LIN {X 0,Y 228.554,Z 405.474,A -85,B 0,C 180,E1 -19981.761,E2 -19981.761} C_VEL
LIN {X 0,Y 228.355,Z 405.527,A -85,B 0,C 180,E1 -19987.07,E2 -19987.07} C_VEL
LIN {X 0,Y 228.163,Z 405.519,A -85,B 0,C 180,E1 -19990.649,E2 -19990.649} C_VEL
LIN {X 0,Y 228.064,Z 405.576,A -85,B 0,C 180,E1 -19994.271,E2 -19994.271} C_VEL
LIN {X 0,Y 228.002,Z 405.55,A -85,B 0,C 180,E1 -19997.952,E2 -19997.952} C_VEL
LIN {X 0,Y 227.929,Z 405.587,A -85,B 0,C 180,E1 -20002.328,E2 -20002.328} C_VEL
LIN {X 0,Y 227.94,Z 405.561,A -85,B 0,C 180,E1 -20006.601,E2 -20006.601} C_VEL
LIN {X 0,Y 227.895,Z 405.594,A -85,B 0,C 180,E1 -20010.29,E2 -20010.29} C_VEL
LIN {X 0,Y 227.887,Z 405.574,A -85,B 0,C 180,E1 -20013.717,E2 -20013.717} C_VEL
LIN {X 0,Y 227.868,Z 405.602,A -85,B 0,C 180,E1 -20018.085,E2 -20018.085} C_VEL
LIN {X 0,Y 227.813,Z 405.604,A -85,B 0,C 180,E1 -20022.74,E2 -20022.74} C_VEL
LIN {X 0,Y 227.812,Z 405.544,A -85,B 0,C 180,E1 -20027.258,E2 -20027.258} C_VEL
LIN {X 0,Y 227.868,Z 405.602,A -85,B 0,C 180,E1 -20031.913,E2 -20031.913} C_VEL
LIN {X 0,Y 227.951,Z 405.9,A -85,B 0,C 180,E1 -20032.927,E2 -20032.927} C_VEL
LIN {X 0,Y 228.325,Z 407.207,A -85,B 0,C 180,E1 -20033.243,E2 -20033.243} C_VEL
LIN {X 0,Y 229.944,Z 409.725,A -85,B 0,C 180,E1 -20033.653,E2 -20033.653} C_VEL
LIN {X 0,Y 238.782,Z 424.968,A -85,B 0,C 180,E1 -20035.756,E2 -20035.756} C_VEL
LIN {X 0,Y 245.467,Z 437.776,A -85,B 0,C 180,E1 -20037.257,E2 -20037.257} C_VEL
LIN {X 0,Y 252.292,Z 450.513,A -85,B 0,C 180,E1 -20038.673,E2 -20038.673} C_VEL
LIN {X 0,Y 260.836,Z 463.188,A -85,B 0,C 180,E1 -20040.213,E2 -20040.213} C_VEL
LIN {X 0,Y 271.083,Z 475.491,A -85,B 0,C 180,E1 -20041.818,E2 -20041.818} C_VEL
LIN {X 0,Y 285.472,Z 490.143,A -85,B 0,C 180,E1 -20043.771,E2 -20043.771} C_VEL
LIN {X 0,Y 299.445,Z 502.11,A -85,B 0,C 180,E1 -20045.429,E2 -20045.429} C_VEL
LIN {X 0,Y 307.354,Z 508.55,A -85,B 0,C 180,E1 -20046.449,E2 -20046.449} C_VEL
LIN {X 0,Y 315.809,Z 515.11,A -85,B 0,C 180,E1 -20047.77,E2 -20047.77} C_VEL
LIN {X 0,Y 323.821,Z 521.078,A -85,B 0,C 180,E1 -20049.216,E2 -20049.216} C_VEL
LIN {X 0,Y 332.128,Z 527.32,A -85,B 0,C 180,E1 -20050.94,E2 -20050.94} C_VEL
LIN {X 0,Y 338.952,Z 531.879,A -85,B 0,C 180,E1 -20052.51,E2 -20052.51} C_VEL
LIN {X 0,Y 345.131,Z 536.469,A -85,B 0,C 180,E1 -20054.129,E2 -20054.129} C_VEL
LIN {X 0,Y 348.902,Z 539.004,A -85,B 0,C 180,E1 -20055.208,E2 -20055.208} C_VEL
LIN {X 0,Y 353.812,Z 541.898,A -85,B 0,C 180,E1 -20056.731,E2 -20056.731} C_VEL
LIN {X 0,Y 357.273,Z 544.165,A -85,B 0,C 180,E1 -20057.966,E2 -20057.966} C_VEL
LIN {X 0,Y 361.925,Z 547.614,A -85,B 0,C 180,E1 -20059.935,E2 -20059.935} C_VEL
LIN {X 0,Y 364.433,Z 549.121,A -85,B 0,C 180,E1 -20061.125,E2 -20061.125} C_VEL
LIN {X 0,Y 368.054,Z 551.052,A -85,B 0,C 180,E1 -20063.181,E2 -20063.181} C_VEL
LIN {X 0,Y 369.976,Z 551.886,A -85,B 0,C 180,E1 -20064.55,E2 -20064.55} C_VEL
LIN {X 0,Y 371.247,Z 552.35,A -85,B 0,C 180,E1 -20065.657,E2 -20065.657} C_VEL
LIN {X 0,Y 372.237,Z 552.641,A -85,B 0,C 180,E1 -20066.753,E2 -20066.753} C_VEL
LIN {X 0,Y 372.88,Z 552.99,A -85,B 0,C 180,E1 -20067.839,E2 -20067.839} C_VEL
LIN {X 0,Y 373.24,Z 553.258,A -85,B 0,C 180,E1 -20068.921,E2 -20068.921} C_VEL
LIN {X 0,Y 373.406,Z 553.214,A -85,B 0,C 180,E1 -20070,E2 -20070} C_VEL
LIN {X 0,Y 373.262,Z 553.193,A -85,B 0,C 180,E1 -20071.079,E2 -20071.079} C_VEL
LIN {X 0,Y 372.799,Z 552.913,A -85,B 0,C 180,E1 -20072.373,E2 -20072.373} C_VEL
LIN {X 0,Y 371.244,Z 552.366,A -85,B 0,C 180,E1 -20074.342,E2 -20074.342} C_VEL
LIN {X 0,Y 369.973,Z 551.918,A -85,B 0,C 180,E1 -20075.45,E2 -20075.45} C_VEL
LIN {X 0,Y 368.059,Z 551.052,A -85,B 0,C 180,E1 -20076.825,E2 -20076.825} C_VEL
LIN {X 0,Y 364.441,Z 549.115,A -85,B 0,C 180,E1 -20078.874,E2 -20078.874} C_VEL
LIN {X 0,Y 360.218,Z 546.455,A -85,B 0,C 180,E1 -20080.812,E2 -20080.812} C_VEL
LIN {X 0,Y 355.924,Z 543.055,A -85,B 0,C 180,E1 -20082.544,E2 -20082.544} C_VEL
LIN {X 0,Y 351.923,Z 540.864,A -85,B 0,C 180,E1 -20083.865,E2 -20083.865} C_VEL
LIN {X 0,Y 345.74,Z 536.848,A -85,B 0,C 180,E1 -20085.708,E2 -20085.708} C_VEL
LIN {X 0,Y 338.968,Z 531.895,A -85,B 0,C 180,E1 -20087.498,E2 -20087.498} C_VEL
LIN {X 0,Y 331.843,Z 527.13,A -85,B 0,C 180,E1 -20089.121,E2 -20089.121} C_VEL
LIN {X 0,Y 323.739,Z 521.021,A -85,B 0,C 180,E1 -20090.798,E2 -20090.798} C_VEL
LIN {X 0,Y 315.796,Z 515.105,A -85,B 0,C 180,E1 -20092.23,E2 -20092.23} C_VEL
LIN {X 0,Y 307.554,Z 508.722,A -85,B 0,C 180,E1 -20093.524,E2 -20093.524} C_VEL
LIN {X 0,Y 300.572,Z 502.979,A -85,B 0,C 180,E1 -20094.436,E2 -20094.436} C_VEL
LIN {X 0,Y 291.164,Z 495.16,A -85,B 0,C 180,E1 -20095.539,E2 -20095.539} C_VEL
LIN {X 0,Y 280.858,Z 485.585,A -85,B 0,C 180,E1 -20096.826,E2 -20096.826} C_VEL
LIN {X 0,Y 268.674,Z 472.809,A -85,B 0,C 180,E1 -20098.54,E2 -20098.54} C_VEL
LIN {X 0,Y 260.028,Z 462.067,A -85,B 0,C 180,E1 -20099.925,E2 -20099.925} C_VEL
LIN {X 0,Y 252.005,Z 450.092,A -85,B 0,C 180,E1 -20101.38,E2 -20101.38} C_VEL
LIN {X 0,Y 245.113,Z 437.01,A -85,B 0,C 180,E1 -20102.822,E2 -20102.822} C_VEL
LIN {X 0,Y 237.86,Z 423.227,A -85,B 0,C 180,E1 -20104.459,E2 -20104.459} C_VEL
LIN {X 0,Y 229.958,Z 409.757,A -85,B 0,C 180,E1 -20106.343,E2 -20106.343} C_VEL
LIN {X 0,Y 228.326,Z 407.225,A -85,B 0,C 180,E1 -20106.756,E2 -20106.756} C_VEL
LIN {X 0,Y 227.923,Z 405.904,A -85,B 0,C 180,E1 -20107.08,E2 -20107.08} C_VEL
LIN {X 0,Y 227.865,Z 405.602,A -85,B 0,C 180,E1 -20108.086,E2 -20108.086} C_VEL
LIN {X 0,Y 227.81,Z 405.544,A -85,B 0,C 180,E1 -20112.741,E2 -20112.741} C_VEL
LIN {X 0,Y 227.893,Z 405.594,A -85,B 0,C 180,E1 -20117.278,E2 -20117.278} C_VEL
LIN {X 0,Y 227.866,Z 405.603,A -85,B 0,C 180,E1 -20121.915,E2 -20121.915} C_VEL
LIN {X 0,Y 227.885,Z 405.575,A -85,B 0,C 180,E1 -20126.373,E2 -20126.373} C_VEL
LIN {X 0,Y 227.914,Z 405.582,A -85,B 0,C 180,E1 -20130.438,E2 -20130.438} C_VEL
LIN {X 0,Y 227.923,Z 405.575,A -85,B 0,C 180,E1 -20134.426,E2 -20134.426} C_VEL
LIN {X 0,Y 227.957,Z 405.575,A -85,B 0,C 180,E1 -20138.288,E2 -20138.288} C_VEL
LIN {X 0,Y 228.03,Z 405.558,A -85,B 0,C 180,E1 -20142.827,E2 -20142.827} C_VEL
LIN {X 0,Y 228.09,Z 405.55,A -85,B 0,C 180,E1 -20147.545,E2 -20147.545} C_VEL
LIN {X 0,Y 228.301,Z 405.507,A -85,B 0,C 180,E1 -20151.147,E2 -20151.147} C_VEL
LIN {X 0,Y 228.351,Z 405.527,A -85,B 0,C 180,E1 -20152.929,E2 -20152.929} C_VEL
LIN {X 0,Y 228.551,Z 405.475,A -85,B 0,C 180,E1 -20158.239,E2 -20158.239} C_VEL
LIN {X 0,Y 228.551,Z 405.487,A -85,B 0,C 180,E1 -20161.763,E2 -20161.763} C_VEL
LIN {X 0,Y 228.352,Z 405.514,A -85,B 0,C 180,E1 -20167.073,E2 -20167.073} C_VEL
LIN {X 0,Y 228.16,Z 405.522,A -85,B 0,C 180,E1 -20170.651,E2 -20170.651} C_VEL
LIN {X 0,Y 228.062,Z 405.574,A -85,B 0,C 180,E1 -20174.273,E2 -20174.273} C_VEL
LIN {X 0,Y 228,Z 405.541,A -85,B 0,C 180,E1 -20177.954,E2 -20177.954} C_VEL
LIN {X 0,Y 227.928,Z 405.59,A -85,B 0,C 180,E1 -20182.331,E2 -20182.331} C_VEL
LIN {X 0,Y 227.941,Z 405.556,A -85,B 0,C 180,E1 -20186.604,E2 -20186.604} C_VEL
LIN {X 0,Y 227.908,Z 405.597,A -85,B 0,C 180,E1 -20190.298,E2 -20190.298} C_VEL
LIN {X 0,Y 227.888,Z 405.571,A -85,B 0,C 180,E1 -20193.72,E2 -20193.72} C_VEL
LIN {X 0,Y 227.871,Z 405.595,A -85,B 0,C 180,E1 -20198.087,E2 -20198.087} C_VEL
LIN {X 0,Y 227.917,Z 405.593,A -85,B 0,C 180,E1 -20202.719,E2 -20202.719} C_VEL
LIN {X 0,Y 227.899,Z 405.809,A -85,B 0,C 180,E1 -20207.645,E2 -20207.645} C_VEL
LIN {X 0,Y 229.638,Z 413.101,A -85,B 0,C 180,E1 -20212.26,E2 -20212.26} C_VEL
LIN {X 0,Y 230.148,Z 415.394,A -85,B 0,C 180,E1 -20213.453,E2 -20213.453} C_VEL
LIN {X 0,Y 232.024,Z 419.408,A -85,B 0,C 180,E1 -20214.009,E2 -20214.009} C_VEL
LIN {X 0,Y 240.511,Z 437.365,A -85,B 0,C 180,E1 -20216.088,E2 -20216.088} C_VEL
LIN {X 0,Y 243.824,Z 445.896,A -85,B 0,C 180,E1 -20216.9,E2 -20216.9} C_VEL
LIN {X 0,Y 247.873,Z 469.061,A -85,B 0,C 180,E1 -20218.278,E2 -20218.278} C_VEL
LIN {X 0,Y 248.138,Z 472.35,A -85,B 0,C 180,E1 -20218.425,E2 -20218.425} C_VEL
LIN {X 0,Y 248.05,Z 474.394,A -85,B 0,C 180,E1 -20218.48,E2 -20218.48} C_VEL
LIN {X 0,Y 247.227,Z 480.242,A -85,B 0,C 180,E1 -20218.559,E2 -20218.559} C_VEL
LIN {X 0,Y 241.567,Z 499.251,A -85,B 0,C 180,E1 -20218.392,E2 -20218.392} C_VEL
LIN {X 0,Y 240.81,Z 505.095,A -85,B 0,C 180,E1 -20218.482,E2 -20218.482} C_VEL
LIN {X 0,Y 239.876,Z 524.739,A -85,B 0,C 180,E1 -20219.12,E2 -20219.12} C_VEL
LIN {X 0,Y 238.394,Z 538.868,A -85,B 0,C 180,E1 -20219.924,E2 -20219.924} C_VEL
LIN {X 0,Y 236.942,Z 548.514,A -85,B 0,C 180,E1 -20220.699,E2 -20220.699} C_VEL
LIN {X 0,Y 235.223,Z 558.034,A -85,B 0,C 180,E1 -20221.686,E2 -20221.686} C_VEL
LIN {X 0,Y 233.004,Z 568.622,A -85,B 0,C 180,E1 -20223.101,E2 -20223.101} C_VEL
LIN {X 0,Y 230.914,Z 577.345,A -85,B 0,C 180,E1 -20224.54,E2 -20224.54} C_VEL
LIN {X 0,Y 229.001,Z 584.763,A -85,B 0,C 180,E1 -20226.007,E2 -20226.007} C_VEL
LIN {X 0,Y 226.579,Z 593.556,A -85,B 0,C 180,E1 -20228.149,E2 -20228.149} C_VEL
LIN {X 0,Y 225.092,Z 599.552,A -85,B 0,C 180,E1 -20229.914,E2 -20229.914} C_VEL
LIN {X 0,Y 223.198,Z 605.86,A -85,B 0,C 180,E1 -20232.122,E2 -20232.122} C_VEL
LIN {X 0,Y 221.656,Z 611.133,A -85,B 0,C 180,E1 -20234.366,E2 -20234.366} C_VEL
LIN {X 0,Y 220.226,Z 616.228,A -85,B 0,C 180,E1 -20237.093,E2 -20237.093} C_VEL
LIN {X 0,Y 219.318,Z 620.197,A -85,B 0,C 180,E1 -20239.849,E2 -20239.849} C_VEL
LIN {X 0,Y 218.762,Z 623.136,A -85,B 0,C 180,E1 -20242.617,E2 -20242.617} C_VEL
LIN {X 0,Y 218.572,Z 624.64,A -85,B 0,C 180,E1 -20244.465,E2 -20244.465} C_VEL
LIN {X 0,Y 218.525,Z 626.171,A -85,B 0,C 180,E1 -20248.158,E2 -20248.158} C_VEL
LIN {X 0,Y 218.622,Z 626.454,A -85,B 0,C 180,E1 -20250.001,E2 -20250.001} C_VEL
LIN {X 0,Y 218.501,Z 625.572,A -85,B 0,C 180,E1 -20253.689,E2 -20253.689} C_VEL
LIN {X 0,Y 218.568,Z 624.64,A -85,B 0,C 180,E1 -20255.536,E2 -20255.536} C_VEL
LIN {X 0,Y 219.088,Z 621.286,A -85,B 0,C 180,E1 -20259.23,E2 -20259.23} C_VEL
LIN {X 0,Y 219.88,Z 617.656,A -85,B 0,C 180,E1 -20261.991,E2 -20261.991} C_VEL
LIN {X 0,Y 221.07,Z 612.92,A -85,B 0,C 180,E1 -20264.734,E2 -20264.734} C_VEL
LIN {X 0,Y 222.916,Z 606.951,A -85,B 0,C 180,E1 -20267.429,E2 -20267.429} C_VEL
LIN {X 0,Y 224.294,Z 602.171,A -85,B 0,C 180,E1 -20269.209,E2 -20269.209} C_VEL
LIN {X 0,Y 226.087,Z 595.69,A -85,B 0,C 180,E1 -20271.248,E2 -20271.248} C_VEL
LIN {X 0,Y 228.023,Z 588.459,A -85,B 0,C 180,E1 -20273.14,E2 -20273.14} C_VEL
LIN {X 0,Y 230.132,Z 580.635,A -85,B 0,C 180,E1 -20274.829,E2 -20274.829} C_VEL
LIN {X 0,Y 232.114,Z 572.554,A -85,B 0,C 180,E1 -20276.284,E2 -20276.284} C_VEL
LIN {X 0,Y 234.273,Z 562.796,A -85,B 0,C 180,E1 -20277.71,E2 -20277.71} C_VEL
LIN {X 0,Y 235.869,Z 554.406,A -85,B 0,C 180,E1 -20278.716,E2 -20278.716} C_VEL
LIN {X 0,Y 237.601,Z 543.903,A -85,B 0,C 180,E1 -20279.699,E2 -20279.699} C_VEL
LIN {X 0,Y 239.038,Z 533.59,A -85,B 0,C 180,E1 -20280.413,E2 -20280.413} C_VEL
LIN {X 0,Y 239.996,Z 523.576,A -85,B 0,C 180,E1 -20280.917,E2 -20280.917} C_VEL
LIN {X 0,Y 240.908,Z 502.246,A -85,B 0,C 180,E1 -20281.601,E2 -20281.601} C_VEL
LIN {X 0,Y 242.123,Z 471.972,A -85,B 0,C 180,E1 -20282.46,E2 -20282.46} C_VEL
LIN {X 0,Y 238.762,Z 452.033,A -85,B 0,C 180,E1 -20283.673,E2 -20283.673} C_VEL
LIN {X 0,Y 237.532,Z 446.723,A -85,B 0,C 180,E1 -20284.058,E2 -20284.058} C_VEL
LIN {X 0,Y 230.678,Z 430.987,A -85,B 0,C 180,E1 -20285.797,E2 -20285.797} C_VEL
LIN {X 0,Y 224.359,Z 418.419,A -85,B 0,C 180,E1 -20287.454,E2 -20287.454} C_VEL
LIN {X 0,Y 222.822,Z 414.942,A -85,B 0,C 180,E1 -20288.007,E2 -20288.007} C_VEL
LIN {X 0,Y 221.346,Z 408.913,A -85,B 0,C 180,E1 -20291.819,E2 -20291.819} C_VEL
LIN {X 0,Y 220.803,Z 406.564,A -85,B 0,C 180,E1 -20293.486,E2 -20293.486} C_VEL
LIN {X 0,Y 220.863,Z 406.473,A -85,B 0,C 180,E1 -20298.068,E2 -20298.068} C_VEL
LIN {X 0,Y 220.838,Z 406.477,A -85,B 0,C 180,E1 -20302.794,E2 -20302.794} C_VEL
LIN {X 0,Y 220.827,Z 406.456,A -85,B 0,C 180,E1 -20307.244,E2 -20307.244} C_VEL
LIN {X 0,Y 220.839,Z 406.453,A -85,B 0,C 180,E1 -20311.486,E2 -20311.486} C_VEL
LIN {X 0,Y 220.869,Z 406.457,A -85,B 0,C 180,E1 -20315.564,E2 -20315.564} C_VEL
LIN {X 0,Y 220.894,Z 406.441,A -85,B 0,C 180,E1 -20319.513,E2 -20319.513} C_VEL
LIN {X 0,Y 221.018,Z 406.423,A -85,B 0,C 180,E1 -20323.369,E2 -20323.369} C_VEL
LIN {X 0,Y 221.113,Z 406.402,A -85,B 0,C 180,E1 -20329.005,E2 -20329.005} C_VEL
LIN {X 0,Y 221.291,Z 406.388,A -85,B 0,C 180,E1 -20332.701,E2 -20332.701} C_VEL
LIN {X 0,Y 221.513,Z 406.363,A -85,B 0,C 180,E1 -20338.181,E2 -20338.181} C_VEL
LIN {X 0,Y 221.512,Z 406.351,A -85,B 0,C 180,E1 -20341.817,E2 -20341.817} C_VEL
LIN {X 0,Y 221.306,Z 406.402,A -85,B 0,C 180,E1 -20347.297,E2 -20347.297} C_VEL
LIN {X 0,Y 221.112,Z 406.399,A -85,B 0,C 180,E1 -20350.993,E2 -20350.993} C_VEL
LIN {X 0,Y 221.016,Z 406.438,A -85,B 0,C 180,E1 -20356.629,E2 -20356.629} C_VEL
LIN {X 0,Y 220.891,Z 406.435,A -85,B 0,C 180,E1 -20360.485,E2 -20360.485} C_VEL
LIN {X 0,Y 220.866,Z 406.47,A -85,B 0,C 180,E1 -20364.434,E2 -20364.434} C_VEL
LIN {X 0,Y 220.825,Z 406.449,A -85,B 0,C 180,E1 -20368.514,E2 -20368.514} C_VEL
LIN {X 0,Y 220.821,Z 406.465,A -85,B 0,C 180,E1 -20372.754,E2 -20372.754} C_VEL
LIN {X 0,Y 220.836,Z 406.477,A -85,B 0,C 180,E1 -20377.287,E2 -20377.287} C_VEL
LIN {X 0,Y 220.773,Z 406.469,A -85,B 0,C 180,E1 -20381.95,E2 -20381.95} C_VEL
LIN {X 0,Y 220.773,Z 406.442,A -85,B 0,C 180,E1 -20385.546,E2 -20385.546} C_VEL
LIN {X 0,Y 220.807,Z 406.439,A -85,B 0,C 180,E1 -20390.463,E2 -20390.463} C_VEL
LIN {X 0,Y 220.871,Z 406.783,A -85,B 0,C 180,E1 -20391.555,E2 -20391.555} C_VEL
LIN {X 0,Y 221.24,Z 408.118,A -85,B 0,C 180,E1 -20391.887,E2 -20391.887} C_VEL
LIN {X 0,Y 222.989,Z 410.766,A -85,B 0,C 180,E1 -20392.359,E2 -20392.359} C_VEL
LIN {X 0,Y 230.451,Z 423.139,A -85,B 0,C 180,E1 -20394.254,E2 -20394.254} C_VEL
LIN {X 0,Y 237.954,Z 436.997,A -85,B 0,C 180,E1 -20396.05,E2 -20396.05} C_VEL
LIN {X 0,Y 246.373,Z 453.364,A -85,B 0,C 180,E1 -20397.922,E2 -20397.922} C_VEL
LIN {X 0,Y 254.155,Z 465.309,A -85,B 0,C 180,E1 -20399.409,E2 -20399.409} C_VEL
LIN {X 0,Y 261.763,Z 475.126,A -85,B 0,C 180,E1 -20400.699,E2 -20400.699} C_VEL
LIN {X 0,Y 274.478,Z 489.059,A -85,B 0,C 180,E1 -20402.593,E2 -20402.593} C_VEL
LIN {X 0,Y 285.936,Z 499.796,A -85,B 0,C 180,E1 -20404.082,E2 -20404.082} C_VEL
LIN {X 0,Y 296.699,Z 508.846,A -85,B 0,C 180,E1 -20405.365,E2 -20405.365} C_VEL
LIN {X 0,Y 304.926,Z 515.571,A -85,B 0,C 180,E1 -20406.473,E2 -20406.473} C_VEL
LIN {X 0,Y 312.987,Z 521.784,A -85,B 0,C 180,E1 -20407.749,E2 -20407.749} C_VEL
LIN {X 0,Y 321.067,Z 527.71,A -85,B 0,C 180,E1 -20409.205,E2 -20409.205} C_VEL
LIN {X 0,Y 327.826,Z 532.846,A -85,B 0,C 180,E1 -20410.608,E2 -20410.608} C_VEL
LIN {X 0,Y 332.996,Z 536.412,A -85,B 0,C 180,E1 -20411.755,E2 -20411.755} C_VEL
LIN {X 0,Y 338.549,Z 540.283,A -85,B 0,C 180,E1 -20413.104,E2 -20413.104} C_VEL
LIN {X 0,Y 343.97,Z 544.192,A -85,B 0,C 180,E1 -20414.596,E2 -20414.596} C_VEL
LIN {X 0,Y 348.701,Z 547.147,A -85,B 0,C 180,E1 -20416.004,E2 -20416.004} C_VEL
LIN {X 0,Y 352.905,Z 549.493,A -85,B 0,C 180,E1 -20417.371,E2 -20417.371} C_VEL
LIN {X 0,Y 357.622,Z 553.083,A -85,B 0,C 180,E1 -20419.292,E2 -20419.292} C_VEL
LIN {X 0,Y 361.373,Z 555.513,A -85,B 0,C 180,E1 -20421.049,E2 -20421.049} C_VEL
LIN {X 0,Y 363.554,Z 556.729,A -85,B 0,C 180,E1 -20422.223,E2 -20422.223} C_VEL
LIN {X 0,Y 365.443,Z 557.658,A -85,B 0,C 180,E1 -20423.374,E2 -20423.374} C_VEL
LIN {X 0,Y 367.106,Z 558.35,A -85,B 0,C 180,E1 -20424.557,E2 -20424.557} C_VEL
LIN {X 0,Y 368.317,Z 558.822,A -85,B 0,C 180,E1 -20425.622,E2 -20425.622} C_VEL
LIN {X 0,Y 369.338,Z 559.106,A -85,B 0,C 180,E1 -20426.727,E2 -20426.727} C_VEL
LIN {X 0,Y 369.982,Z 559.47,A -85,B 0,C 180,E1 -20427.822,E2 -20427.822} C_VEL
LIN {X 0,Y 370.34,Z 559.737,A -85,B 0,C 180,E1 -20428.912,E2 -20428.912} C_VEL
LIN {X 0,Y 370.526,Z 559.673,A -85,B 0,C 180,E1 -20430,E2 -20430} C_VEL
LIN {X 0,Y 370.373,Z 559.651,A -85,B 0,C 180,E1 -20431.087,E2 -20431.087} C_VEL
LIN {X 0,Y 369.987,Z 559.435,A -85,B 0,C 180,E1 -20432.177,E2 -20432.177} C_VEL
LIN {X 0,Y 369.329,Z 559.095,A -85,B 0,C 180,E1 -20433.272,E2 -20433.272} C_VEL
LIN {X 0,Y 368.306,Z 558.822,A -85,B 0,C 180,E1 -20434.377,E2 -20434.377} C_VEL
LIN {X 0,Y 367.014,Z 558.361,A -85,B 0,C 180,E1 -20435.494,E2 -20435.494} C_VEL
LIN {X 0,Y 365.444,Z 557.664,A -85,B 0,C 180,E1 -20436.626,E2 -20436.626} C_VEL
LIN {X 0,Y 362.347,Z 556.045,A -85,B 0,C 180,E1 -20438.44,E2 -20438.44} C_VEL
LIN {X 0,Y 358.851,Z 553.978,A -85,B 0,C 180,E1 -20440.152,E2 -20440.152} C_VEL
LIN {X 0,Y 354.946,Z 551.149,A -85,B 0,C 180,E1 -20441.817,E2 -20441.817} C_VEL
LIN {X 0,Y 352.841,Z 549.405,A -85,B 0,C 180,E1 -20442.656,E2 -20442.656} C_VEL
LIN {X 0,Y 347.995,Z 546.721,A -85,B 0,C 180,E1 -20444.216,E2 -20444.216} C_VEL
LIN {X 0,Y 343.051,Z 543.53,A -85,B 0,C 180,E1 -20445.664,E2 -20445.664} C_VEL
LIN {X 0,Y 338.092,Z 539.928,A -85,B 0,C 180,E1 -20447.021,E2 -20447.021} C_VEL
LIN {X 0,Y 330.726,Z 534.904,A -85,B 0,C 180,E1 -20448.765,E2 -20448.765} C_VEL
LIN {X 0,Y 323.611,Z 529.586,A -85,B 0,C 180,E1 -20450.289,E2 -20450.289} C_VEL
LIN {X 0,Y 314.843,Z 523.218,A -85,B 0,C 180,E1 -20451.931,E2 -20451.931} C_VEL
LIN {X 0,Y 306.174,Z 516.524,A -85,B 0,C 180,E1 -20453.342,E2 -20453.342} C_VEL
LIN {X 0,Y 298,Z 509.994,A -85,B 0,C 180,E1 -20454.471,E2 -20454.471} C_VEL
LIN {X 0,Y 286.124,Z 499.956,A -85,B 0,C 180,E1 -20455.895,E2 -20455.895} C_VEL
LIN {X 0,Y 276.695,Z 491.195,A -85,B 0,C 180,E1 -20457.106,E2 -20457.106} C_VEL
LIN {X 0,Y 263.991,Z 477.806,A -85,B 0,C 180,E1 -20458.946,E2 -20458.946} C_VEL
LIN {X 0,Y 255.164,Z 466.754,A -85,B 0,C 180,E1 -20460.41,E2 -20460.41} C_VEL
LIN {X 0,Y 247.279,Z 454.927,A -85,B 0,C 180,E1 -20461.893,E2 -20461.893} C_VEL
LIN {X 0,Y 240.22,Z 441.558,A -85,B 0,C 180,E1 -20463.424,E2 -20463.424} C_VEL
LIN {X 0,Y 233.03,Z 427.701,A -85,B 0,C 180,E1 -20465.119,E2 -20465.119} C_VEL
LIN {X 0,Y 225.322,Z 414.513,A -85,B 0,C 180,E1 -20467.035,E2 -20467.035} C_VEL
LIN {X 0,Y 222.666,Z 410.45,A -85,B 0,C 180,E1 -20467.718,E2 -20467.718} C_VEL
LIN {X 0,Y 221.04,Z 407.573,A -85,B 0,C 180,E1 -20468.198,E2 -20468.198} C_VEL
LIN {X 0,Y 220.855,Z 406.692,A -85,B 0,C 180,E1 -20468.515,E2 -20468.515} C_VEL
LIN {X 0,Y 220.77,Z 406.418,A -85,B 0,C 180,E1 -20471.951,E2 -20471.951} C_VEL
LIN {X 0,Y 220.852,Z 406.474,A -85,B 0,C 180,E1 -20477.045,E2 -20477.045} C_VEL
LIN {X 0,Y 220.807,Z 406.464,A -85,B 0,C 180,E1 -20480.465,E2 -20480.465} C_VEL
LIN {X 0,Y 220.83,Z 406.477,A -85,B 0,C 180,E1 -20482.795,E2 -20482.795} C_VEL
LIN {X 0,Y 220.819,Z 406.465,A -85,B 0,C 180,E1 -20487.246,E2 -20487.246} C_VEL
LIN {X 0,Y 220.831,Z 406.448,A -85,B 0,C 180,E1 -20491.487,E2 -20491.487} C_VEL
LIN {X 0,Y 220.862,Z 406.47,A -85,B 0,C 180,E1 -20495.566,E2 -20495.566} C_VEL
LIN {X 0,Y 220.887,Z 406.435,A -85,B 0,C 180,E1 -20499.515,E2 -20499.515} C_VEL
LIN {X 0,Y 221.012,Z 406.439,A -85,B 0,C 180,E1 -20503.371,E2 -20503.371} C_VEL
LIN {X 0,Y 221.108,Z 406.399,A -85,B 0,C 180,E1 -20509.007,E2 -20509.007} C_VEL
LIN {X 0,Y 221.302,Z 406.402,A -85,B 0,C 180,E1 -20512.703,E2 -20512.703} C_VEL
LIN {X 0,Y 221.509,Z 406.352,A -85,B 0,C 180,E1 -20518.183,E2 -20518.183} C_VEL
LIN {X 0,Y 221.509,Z 406.363,A -85,B 0,C 180,E1 -20521.819,E2 -20521.819} C_VEL
LIN {X 0,Y 221.287,Z 406.389,A -85,B 0,C 180,E1 -20527.3,E2 -20527.3} C_VEL
LIN {X 0,Y 221.109,Z 406.403,A -85,B 0,C 180,E1 -20530.995,E2 -20530.995} C_VEL
LIN {X 0,Y 221.014,Z 406.424,A -85,B 0,C 180,E1 -20536.631,E2 -20536.631} C_VEL
LIN {X 0,Y 220.89,Z 406.442,A -85,B 0,C 180,E1 -20540.487,E2 -20540.487} C_VEL
LIN {X 0,Y 220.866,Z 406.458,A -85,B 0,C 180,E1 -20544.436,E2 -20544.436} C_VEL
LIN {X 0,Y 220.835,Z 406.454,A -85,B 0,C 180,E1 -20548.515,E2 -20548.515} C_VEL
LIN {X 0,Y 220.823,Z 406.456,A -85,B 0,C 180,E1 -20552.756,E2 -20552.756} C_VEL
LIN {X 0,Y 220.838,Z 406.477,A -85,B 0,C 180,E1 -20557.289,E2 -20557.289} C_VEL
LIN {X 0,Y 220.86,Z 406.473,A -85,B 0,C 180,E1 -20561.933,E2 -20561.933} C_VEL
LIN {X 0,Y 220.808,Z 406.609,A -85,B 0,C 180,E1 -20566.591,E2 -20566.591} C_VEL
LIN {X 0,Y 222.603,Z 414.108,A -85,B 0,C 180,E1 -20571.575,E2 -20571.575} C_VEL
LIN {X 0,Y 222.982,Z 415.503,A -85,B 0,C 180,E1 -20572.123,E2 -20572.123} C_VEL
LIN {X 0,Y 229.971,Z 429.62,A -85,B 0,C 180,E1 -20574.026,E2 -20574.026} C_VEL
LIN {X 0,Y 235.849,Z 442.572,A -85,B 0,C 180,E1 -20575.517,E2 -20575.517} C_VEL
LIN {X 0,Y 238.132,Z 448.621,A -85,B 0,C 180,E1 -20576.106,E2 -20576.106} C_VEL
LIN {X 0,Y 241.842,Z 470.092,A -85,B 0,C 180,E1 -20577.433,E2 -20577.433} C_VEL
LIN {X 0,Y 242.016,Z 474.614,A -85,B 0,C 180,E1 -20577.614,E2 -20577.614} C_VEL
LIN {X 0,Y 240.81,Z 505.095,A -85,B 0,C 180,E1 -20578.482,E2 -20578.482} C_VEL
LIN {X 0,Y 239.994,Z 510.941,A -85,B 0,C 180,E1 -20578.56,E2 -20578.56} C_VEL
LIN {X 0,Y 236.928,Z 520.398,A -85,B 0,C 180,E1 -20578.486,E2 -20578.486} C_VEL
LIN {X 0,Y 233.713,Z 529.785,A -85,B 0,C 180,E1 -20578.543,E2 -20578.543} C_VEL
LIN {X 0,Y 232.71,Z 535.508,A -85,B 0,C 180,E1 -20578.823,E2 -20578.823} C_VEL
LIN {X 0,Y 230.777,Z 548.319,A -85,B 0,C 180,E1 -20579.836,E2 -20579.836} C_VEL
LIN {X 0,Y 228.967,Z 557.838,A -85,B 0,C 180,E1 -20580.84,E2 -20580.84} C_VEL
LIN {X 0,Y 226.686,Z 568.427,A -85,B 0,C 180,E1 -20582.288,E2 -20582.288} C_VEL
LIN {X 0,Y 224.494,Z 577.149,A -85,B 0,C 180,E1 -20583.757,E2 -20583.757} C_VEL
LIN {X 0,Y 222.508,Z 584.567,A -85,B 0,C 180,E1 -20585.261,E2 -20585.261} C_VEL
LIN {X 0,Y 219.973,Z 593.36,A -85,B 0,C 180,E1 -20587.457,E2 -20587.457} C_VEL
LIN {X 0,Y 218.39,Z 599.355,A -85,B 0,C 180,E1 -20589.269,E2 -20589.269} C_VEL
LIN {X 0,Y 216.4,Z 605.664,A -85,B 0,C 180,E1 -20591.54,E2 -20591.54} C_VEL
LIN {X 0,Y 214.802,Z 610.938,A -85,B 0,C 180,E1 -20593.853,E2 -20593.853} C_VEL
LIN {X 0,Y 213.261,Z 616.032,A -85,B 0,C 180,E1 -20596.663,E2 -20596.663} C_VEL
LIN {X 0,Y 212.304,Z 620.001,A -85,B 0,C 180,E1 -20599.51,E2 -20599.51} C_VEL
LIN {X 0,Y 211.689,Z 622.94,A -85,B 0,C 180,E1 -20602.369,E2 -20602.369} C_VEL
LIN {X 0,Y 211.495,Z 624.445,A -85,B 0,C 180,E1 -20604.279,E2 -20604.279} C_VEL
LIN {X 0,Y 211.427,Z 625.976,A -85,B 0,C 180,E1 -20608.096,E2 -20608.096} C_VEL
LIN {X 0,Y 211.539,Z 626.259,A -85,B 0,C 180,E1 -20610.001,E2 -20610.001} C_VEL
LIN {X 0,Y 211.4,Z 625.376,A -85,B 0,C 180,E1 -20613.813,E2 -20613.813} C_VEL
LIN {X 0,Y 211.49,Z 624.444,A -85,B 0,C 180,E1 -20615.722,E2 -20615.722} C_VEL
LIN {X 0,Y 212.063,Z 621.09,A -85,B 0,C 180,E1 -20619.539,E2 -20619.539} C_VEL
LIN {X 0,Y 212.903,Z 617.459,A -85,B 0,C 180,E1 -20622.391,E2 -20622.391} C_VEL
LIN {X 0,Y 214.197,Z 612.724,A -85,B 0,C 180,E1 -20625.218,E2 -20625.218} C_VEL
LIN {X 0,Y 216.109,Z 606.755,A -85,B 0,C 180,E1 -20627.996,E2 -20627.996} C_VEL
LIN {X 0,Y 217.589,Z 601.976,A -85,B 0,C 180,E1 -20629.825,E2 -20629.825} C_VEL
LIN {X 0,Y 219.347,Z 595.818,A -85,B 0,C 180,E1 -20631.831,E2 -20631.831} C_VEL
LIN {X 0,Y 221.493,Z 588.263,A -85,B 0,C 180,E1 -20633.864,E2 -20633.864} C_VEL
LIN {X 0,Y 223.681,Z 580.439,A -85,B 0,C 180,E1 -20635.596,E2 -20635.596} C_VEL
LIN {X 0,Y 225.77,Z 572.359,A -85,B 0,C 180,E1 -20637.082,E2 -20637.082} C_VEL
LIN {X 0,Y 228.016,Z 562.601,A -85,B 0,C 180,E1 -20638.539,E2 -20638.539} C_VEL
LIN {X 0,Y 229.666,Z 554.211,A -85,B 0,C 180,E1 -20639.567,E2 -20639.567} C_VEL
LIN {X 0,Y 231.482,Z 543.708,A -85,B 0,C 180,E1 -20640.567,E2 -20640.567} C_VEL
LIN {X 0,Y 232.929,Z 533.565,A -85,B 0,C 180,E1 -20641.287,E2 -20641.287} C_VEL
LIN {X 0,Y 233.972,Z 522.911,A -85,B 0,C 180,E1 -20641.827,E2 -20641.827} C_VEL
LIN {X 0,Y 234.937,Z 501.147,A -85,B 0,C 180,E1 -20642.534,E2 -20642.534} C_VEL
LIN {X 0,Y 236.111,Z 472.945,A -85,B 0,C 180,E1 -20643.352,E2 -20643.352} C_VEL
LIN {X 0,Y 233.125,Z 454.838,A -85,B 0,C 180,E1 -20644.491,E2 -20644.491} C_VEL
LIN {X 0,Y 232.01,Z 449.701,A -85,B 0,C 180,E1 -20644.869,E2 -20644.869} C_VEL
LIN {X 0,Y 225.376,Z 434.47,A -85,B 0,C 180,E1 -20646.633,E2 -20646.633} C_VEL
LIN {X 0,Y 219.114,Z 421.84,A -85,B 0,C 180,E1 -20648.365,E2 -20648.365} C_VEL
LIN {X 0,Y 215.55,Z 414.931,A -85,B 0,C 180,E1 -20649.47,E2 -20649.47} C_VEL
LIN {X 0,Y 214.836,Z 412.069,A -85,B 0,C 180,E1 -20651.199,E2 -20651.199} C_VEL
LIN {X 0,Y 213.798,Z 407.431,A -85,B 0,C 180,E1 -20654.527,E2 -20654.527} C_VEL
LIN {X 0,Y 213.801,Z 407.339,A -85,B 0,C 180,E1 -20659.117,E2 -20659.117} C_VEL
LIN {X 0,Y 213.758,Z 407.352,A -85,B 0,C 180,E1 -20663.713,E2 -20663.713} C_VEL
LIN {X 0,Y 213.798,Z 407.35,A -85,B 0,C 180,E1 -20668.724,E2 -20668.724} C_VEL
LIN {X 0,Y 213.828,Z 407.314,A -85,B 0,C 180,E1 -20672.602,E2 -20672.602} C_VEL
LIN {X 0,Y 213.854,Z 407.344,A -85,B 0,C 180,E1 -20676.952,E2 -20676.952} C_VEL
LIN {X 0,Y 213.945,Z 407.296,A -85,B 0,C 180,E1 -20682.803,E2 -20682.803} C_VEL
LIN {X 0,Y 213.982,Z 407.326,A -85,B 0,C 180,E1 -20686.707,E2 -20686.707} C_VEL
LIN {X 0,Y 214.168,Z 407.255,A -85,B 0,C 180,E1 -20690.555,E2 -20690.555} C_VEL
LIN {X 0,Y 214.229,Z 407.262,A -85,B 0,C 180,E1 -20692.459,E2 -20692.459} C_VEL
LIN {X 0,Y 214.446,Z 407.243,A -85,B 0,C 180,E1 -20698.121,E2 -20698.121} C_VEL
LIN {X 0,Y 214.546,Z 407.21,A -85,B 0,C 180,E1 -20699.999,E2 -20699.999} C_VEL
LIN {X 0,Y 214.446,Z 407.231,A -85,B 0,C 180,E1 -20701.877,E2 -20701.877} C_VEL
LIN {X 0,Y 214.24,Z 407.276,A -85,B 0,C 180,E1 -20707.539,E2 -20707.539} C_VEL
LIN {X 0,Y 214.044,Z 407.281,A -85,B 0,C 180,E1 -20711.361,E2 -20711.361} C_VEL
LIN {X 0,Y 213.934,Z 407.336,A -85,B 0,C 180,E1 -20715.236,E2 -20715.236} C_VEL
LIN {X 0,Y 213.838,Z 407.306,A -85,B 0,C 180,E1 -20719.186,E2 -20719.186} C_VEL
LIN {X 0,Y 213.846,Z 407.347,A -85,B 0,C 180,E1 -20723.226,E2 -20723.226} C_VEL
LIN {X 0,Y 213.828,Z 407.315,A -85,B 0,C 180,E1 -20727.449,E2 -20727.449} C_VEL
LIN {X 0,Y 213.768,Z 407.357,A -85,B 0,C 180,E1 -20731.736,E2 -20731.736} C_VEL
LIN {X 0,Y 213.751,Z 407.343,A -85,B 0,C 180,E1 -20736.286,E2 -20736.286} C_VEL
LIN {X 0,Y 213.714,Z 407.342,A -85,B 0,C 180,E1 -20741.123,E2 -20741.123} C_VEL
LIN {X 0,Y 213.708,Z 407.365,A -85,B 0,C 180,E1 -20743.677,E2 -20743.677} C_VEL
LIN {X 0,Y 213.706,Z 407.307,A -85,B 0,C 180,E1 -20746.342,E2 -20746.342} C_VEL
LIN {X 0,Y 213.795,Z 407.509,A -85,B 0,C 180,E1 -20749.96,E2 -20749.96} C_VEL
LIN {X 0,Y 214.068,Z 408.664,A -85,B 0,C 180,E1 -20750.37,E2 -20750.37} C_VEL
LIN {X 0,Y 215.545,Z 411.189,A -85,B 0,C 180,E1 -20750.823,E2 -20750.823} C_VEL
LIN {X 0,Y 216.646,Z 412.747,A -85,B 0,C 180,E1 -20751.127,E2 -20751.127} C_VEL
LIN {X 0,Y 223.733,Z 424.176,A -85,B 0,C 180,E1 -20753.038,E2 -20753.038} C_VEL
LIN {X 0,Y 232.167,Z 439.551,A -85,B 0,C 180,E1 -20755.17,E2 -20755.17} C_VEL
LIN {X 0,Y 241.226,Z 457.456,A -85,B 0,C 180,E1 -20757.289,E2 -20757.289} C_VEL
LIN {X 0,Y 249.298,Z 469.969,A -85,B 0,C 180,E1 -20758.895,E2 -20758.895} C_VEL
LIN {X 0,Y 257.182,Z 480.212,A -85,B 0,C 180,E1 -20760.281,E2 -20760.281} C_VEL
LIN {X 0,Y 270.167,Z 494.492,A -85,B 0,C 180,E1 -20762.275,E2 -20762.275} C_VEL
LIN {X 0,Y 281.485,Z 505.169,A -85,B 0,C 180,E1 -20763.8,E2 -20763.8} C_VEL
LIN {X 0,Y 291.896,Z 514.058,A -85,B 0,C 180,E1 -20765.147,E2 -20765.147} C_VEL
LIN {X 0,Y 301.582,Z 521.908,A -85,B 0,C 180,E1 -20766.469,E2 -20766.469} C_VEL
LIN {X 0,Y 308.415,Z 527.143,A -85,B 0,C 180,E1 -20767.536,E2 -20767.536} C_VEL
LIN {X 0,Y 316.31,Z 532.99,A -85,B 0,C 180,E1 -20768.935,E2 -20768.935} C_VEL
LIN {X 0,Y 323.602,Z 538.492,A -85,B 0,C 180,E1 -20770.421,E2 -20770.421} C_VEL
LIN {X 0,Y 330.787,Z 543.399,A -85,B 0,C 180,E1 -20772.012,E2 -20772.012} C_VEL
LIN {X 0,Y 337.012,Z 547.916,A -85,B 0,C 180,E1 -20773.59,E2 -20773.59} C_VEL
LIN {X 0,Y 341.979,Z 551.295,A -85,B 0,C 180,E1 -20774.99,E2 -20774.99} C_VEL
LIN {X 0,Y 346.925,Z 554.257,A -85,B 0,C 180,E1 -20776.5,E2 -20776.5} C_VEL
LIN {X 0,Y 350.604,Z 556.608,A -85,B 0,C 180,E1 -20777.78,E2 -20777.78} C_VEL
LIN {X 0,Y 355.243,Z 560.043,A -85,B 0,C 180,E1 -20779.743,E2 -20779.743} C_VEL
LIN {X 0,Y 357.792,Z 561.608,A -85,B 0,C 180,E1 -20780.959,E2 -20780.959} C_VEL
LIN {X 0,Y 361.225,Z 563.486,A -85,B 0,C 180,E1 -20782.859,E2 -20782.859} C_VEL
LIN {X 0,Y 363.588,Z 564.533,A -85,B 0,C 180,E1 -20784.454,E2 -20784.454} C_VEL
LIN {X 0,Y 364.925,Z 565.069,A -85,B 0,C 180,E1 -20785.582,E2 -20785.582} C_VEL
LIN {X 0,Y 366.043,Z 565.387,A -85,B 0,C 180,E1 -20786.741,E2 -20786.741} C_VEL
LIN {X 0,Y 366.673,Z 565.728,A -85,B 0,C 180,E1 -20787.803,E2 -20787.803} C_VEL
LIN {X 0,Y 367.035,Z 565.997,A -85,B 0,C 180,E1 -20788.903,E2 -20788.903} C_VEL
LIN {X 0,Y 367.232,Z 565.943,A -85,B 0,C 180,E1 -20790,E2 -20790} C_VEL
LIN {X 0,Y 367.068,Z 565.924,A -85,B 0,C 180,E1 -20791.097,E2 -20791.097} C_VEL
LIN {X 0,Y 366.678,Z 565.698,A -85,B 0,C 180,E1 -20792.197,E2 -20792.197} C_VEL
LIN {X 0,Y 365.987,Z 565.373,A -85,B 0,C 180,E1 -20793.302,E2 -20793.302} C_VEL
LIN {X 0,Y 364.911,Z 565.06,A -85,B 0,C 180,E1 -20794.418,E2 -20794.418} C_VEL
LIN {X 0,Y 363.554,Z 564.556,A -85,B 0,C 180,E1 -20795.546,E2 -20795.546} C_VEL
LIN {X 0,Y 361.235,Z 563.482,A -85,B 0,C 180,E1 -20797.153,E2 -20797.153} C_VEL
LIN {X 0,Y 357.787,Z 561.594,A -85,B 0,C 180,E1 -20799.041,E2 -20799.041} C_VEL
LIN {X 0,Y 353.983,Z 559.2,A -85,B 0,C 180,E1 -20800.809,E2 -20800.809} C_VEL
LIN {X 0,Y 349.096,Z 555.454,A -85,B 0,C 180,E1 -20802.794,E2 -20802.794} C_VEL
LIN {X 0,Y 344.817,Z 553.067,A -85,B 0,C 180,E1 -20804.157,E2 -20804.157} C_VEL
LIN {X 0,Y 339.977,Z 549.962,A -85,B 0,C 180,E1 -20805.588,E2 -20805.588} C_VEL
LIN {X 0,Y 334.345,Z 545.933,A -85,B 0,C 180,E1 -20807.114,E2 -20807.114} C_VEL
LIN {X 0,Y 328.766,Z 542.143,A -85,B 0,C 180,E1 -20808.452,E2 -20808.452} C_VEL
LIN {X 0,Y 321.609,Z 537.001,A -85,B 0,C 180,E1 -20810.008,E2 -20810.008} C_VEL
LIN {X 0,Y 316.31,Z 533.01,A -85,B 0,C 180,E1 -20811.066,E2 -20811.066} C_VEL
LIN {X 0,Y 308.379,Z 527.121,A -85,B 0,C 180,E1 -20812.47,E2 -20812.47} C_VEL
LIN {X 0,Y 300.19,Z 520.842,A -85,B 0,C 180,E1 -20813.729,E2 -20813.729} C_VEL
LIN {X 0,Y 287.807,Z 510.785,A -85,B 0,C 180,E1 -20815.379,E2 -20815.379} C_VEL
LIN {X 0,Y 273.7,Z 497.988,A -85,B 0,C 180,E1 -20817.233,E2 -20817.233} C_VEL
LIN {X 0,Y 260.031,Z 483.623,A -85,B 0,C 180,E1 -20819.253,E2 -20819.253} C_VEL
LIN {X 0,Y 250.581,Z 471.82,A -85,B 0,C 180,E1 -20820.866,E2 -20820.866} C_VEL
LIN {X 0,Y 242.077,Z 458.952,A -85,B 0,C 180,E1 -20822.529,E2 -20822.529} C_VEL
LIN {X 0,Y 234.855,Z 445.03,A -85,B 0,C 180,E1 -20824.173,E2 -20824.173} C_VEL
LIN {X 0,Y 228.092,Z 431.873,A -85,B 0,C 180,E1 -20825.843,E2 -20825.843} C_VEL
LIN {X 0,Y 220.748,Z 419.211,A -85,B 0,C 180,E1 -20827.752,E2 -20827.752} C_VEL
LIN {X 0,Y 216.385,Z 412.199,A -85,B 0,C 180,E1 -20828.952,E2 -20828.952} C_VEL
LIN {X 0,Y 214.254,Z 409.179,A -85,B 0,C 180,E1 -20829.554,E2 -20829.554} C_VEL
LIN {X 0,Y 213.827,Z 407.784,A -85,B 0,C 180,E1 -20829.87,E2 -20829.87} C_VEL
LIN {X 0,Y 213.743,Z 407.361,A -85,B 0,C 180,E1 -20830.402,E2 -20830.402} C_VEL
LIN {X 0,Y 213.707,Z 407.307,A -85,B 0,C 180,E1 -20833.677,E2 -20833.677} C_VEL
LIN {X 0,Y 213.772,Z 407.357,A -85,B 0,C 180,E1 -20836.34,E2 -20836.34} C_VEL
LIN {X 0,Y 213.733,Z 407.356,A -85,B 0,C 180,E1 -20841.337,E2 -20841.337} C_VEL
LIN {X 0,Y 213.763,Z 407.331,A -85,B 0,C 180,E1 -20846.02,E2 -20846.02} C_VEL
LIN {X 0,Y 213.776,Z 407.34,A -85,B 0,C 180,E1 -20850.455,E2 -20850.455} C_VEL
LIN {X 0,Y 213.796,Z 407.337,A -85,B 0,C 180,E1 -20854.702,E2 -20854.702} C_VEL
LIN {X 0,Y 213.807,Z 407.326,A -85,B 0,C 180,E1 -20858.804,E2 -20858.804} C_VEL
LIN {X 0,Y 213.939,Z 407.31,A -85,B 0,C 180,E1 -20862.804,E2 -20862.804} C_VEL
LIN {X 0,Y 213.976,Z 407.322,A -85,B 0,C 180,E1 -20866.709,E2 -20866.709} C_VEL
LIN {X 0,Y 214.163,Z 407.261,A -85,B 0,C 180,E1 -20870.557,E2 -20870.557} C_VEL
LIN {X 0,Y 214.236,Z 407.276,A -85,B 0,C 180,E1 -20872.461,E2 -20872.461} C_VEL
LIN {X 0,Y 214.442,Z 407.231,A -85,B 0,C 180,E1 -20878.123,E2 -20878.123} C_VEL
LIN {X 0,Y 214.543,Z 407.21,A -85,B 0,C 180,E1 -20880.001,E2 -20880.001} C_VEL
LIN {X 0,Y 214.443,Z 407.243,A -85,B 0,C 180,E1 -20881.879,E2 -20881.879} C_VEL
LIN {X 0,Y 214.225,Z 407.263,A -85,B 0,C 180,E1 -20887.542,E2 -20887.542} C_VEL
LIN {X 0,Y 214.042,Z 407.288,A -85,B 0,C 180,E1 -20891.363,E2 -20891.363} C_VEL
LIN {X 0,Y 213.931,Z 407.327,A -85,B 0,C 180,E1 -20895.238,E2 -20895.238} C_VEL
LIN {X 0,Y 213.837,Z 407.305,A -85,B 0,C 180,E1 -20899.189,E2 -20899.189} C_VEL
LIN {X 0,Y 213.846,Z 407.345,A -85,B 0,C 180,E1 -20903.228,E2 -20903.228} C_VEL
LIN {X 0,Y 213.828,Z 407.315,A -85,B 0,C 180,E1 -20907.451,E2 -20907.451} C_VEL
LIN {X 0,Y 213.778,Z 407.347,A -85,B 0,C 180,E1 -20911.737,E2 -20911.737} C_VEL
LIN {X 0,Y 213.754,Z 407.352,A -85,B 0,C 180,E1 -20916.287,E2 -20916.287} C_VEL
LIN {X 0,Y 213.797,Z 407.342,A -85,B 0,C 180,E1 -20921.107,E2 -20921.107} C_VEL
LIN {X 0,Y 213.817,Z 407.487,A -85,B 0,C 180,E1 -20925.552,E2 -20925.552} C_VEL
LIN {X 0,Y 215.456,Z 414.648,A -85,B 0,C 180,E1 -20930.424,E2 -20930.424} C_VEL
LIN {X 0,Y 216.368,Z 416.936,A -85,B 0,C 180,E1 -20930.856,E2 -20930.856} C_VEL
LIN {X 0,Y 218.844,Z 421.32,A -85,B 0,C 180,E1 -20931.558,E2 -20931.558} C_VEL
LIN {X 0,Y 224.774,Z 433.187,A -85,B 0,C 180,E1 -20933.204,E2 -20933.204} C_VEL
LIN {X 0,Y 230.765,Z 446.592,A -85,B 0,C 180,E1 -20934.802,E2 -20934.802} C_VEL
LIN {X 0,Y 232.529,Z 451.601,A -85,B 0,C 180,E1 -20935.29,E2 -20935.29} C_VEL
LIN {X 0,Y 235.989,Z 472.163,A -85,B 0,C 180,E1 -20936.601,E2 -20936.601} C_VEL
LIN {X 0,Y 234.066,Z 520.802,A -85,B 0,C 180,E1 -20938.081,E2 -20938.081} C_VEL
LIN {X 0,Y 233.166,Z 531.392,A -85,B 0,C 180,E1 -20938.589,E2 -20938.589} C_VEL
LIN {X 0,Y 232.71,Z 535.508,A -85,B 0,C 180,E1 -20938.823,E2 -20938.823} C_VEL
LIN {X 0,Y 231.498,Z 541.145,A -85,B 0,C 180,E1 -20939.129,E2 -20939.129} C_VEL
LIN {X 0,Y 227.481,Z 550.04,A -85,B 0,C 180,E1 -20939.566,E2 -20939.566} C_VEL
LIN {X 0,Y 223.174,Z 558.813,A -85,B 0,C 180,E1 -20940.184,E2 -20940.184} C_VEL
LIN {X 0,Y 221.506,Z 563.832,A -85,B 0,C 180,E1 -20940.775,E2 -20940.775} C_VEL
LIN {X 0,Y 218.462,Z 575.856,A -85,B 0,C 180,E1 -20942.715,E2 -20942.715} C_VEL
LIN {X 0,Y 216.069,Z 584.372,A -85,B 0,C 180,E1 -20944.471,E2 -20944.471} C_VEL
LIN {X 0,Y 213.402,Z 593.164,A -85,B 0,C 180,E1 -20946.723,E2 -20946.723} C_VEL
LIN {X 0,Y 211.72,Z 599.159,A -85,B 0,C 180,E1 -20948.585,E2 -20948.585} C_VEL
LIN {X 0,Y 209.642,Z 605.468,A -85,B 0,C 180,E1 -20950.923,E2 -20950.923} C_VEL
LIN {X 0,Y 207.96,Z 610.742,A -85,B 0,C 180,E1 -20953.307,E2 -20953.307} C_VEL
LIN {X 0,Y 206.314,Z 615.835,A -85,B 0,C 180,E1 -20956.206,E2 -20956.206} C_VEL
LIN {X 0,Y 205.282,Z 619.805,A -85,B 0,C 180,E1 -20959.147,E2 -20959.147} C_VEL
LIN {X 0,Y 204.641,Z 622.745,A -85,B 0,C 180,E1 -20962.105,E2 -20962.105} C_VEL
LIN {X 0,Y 204.404,Z 624.249,A -85,B 0,C 180,E1 -20964.08,E2 -20964.08} C_VEL
LIN {X 0,Y 204.333,Z 625.781,A -85,B 0,C 180,E1 -20968.03,E2 -20968.03} C_VEL
LIN {X 0,Y 204.438,Z 626.064,A -85,B 0,C 180,E1 -20970.001,E2 -20970.001} C_VEL
LIN {X 0,Y 204.3,Z 625.181,A -85,B 0,C 180,E1 -20973.946,E2 -20973.946} C_VEL
LIN {X 0,Y 204.396,Z 624.248,A -85,B 0,C 180,E1 -20975.921,E2 -20975.921} C_VEL
LIN {X 0,Y 205.053,Z 620.895,A -85,B 0,C 180,E1 -20979.868,E2 -20979.868} C_VEL
LIN {X 0,Y 205.941,Z 617.263,A -85,B 0,C 180,E1 -20982.816,E2 -20982.816} C_VEL
LIN {X 0,Y 207.339,Z 612.529,A -85,B 0,C 180,E1 -20985.734,E2 -20985.734} C_VEL
LIN {X 0,Y 209.309,Z 606.558,A -85,B 0,C 180,E1 -20988.602,E2 -20988.602} C_VEL
LIN {X 0,Y 211.329,Z 600.469,A -85,B 0,C 180,E1 -20990.947,E2 -20990.947} C_VEL
LIN {X 0,Y 213.047,Z 594.552,A -85,B 0,C 180,E1 -20992.862,E2 -20992.862} C_VEL
LIN {X 0,Y 214.99,Z 588.067,A -85,B 0,C 180,E1 -20994.633,E2 -20994.633} C_VEL
LIN {X 0,Y 217.301,Z 580.244,A -85,B 0,C 180,E1 -20996.405,E2 -20996.405} C_VEL
LIN {X 0,Y 219.454,Z 572.163,A -85,B 0,C 180,E1 -20997.928,E2 -20997.928} C_VEL
LIN {X 0,Y 221.8,Z 562.405,A -85,B 0,C 180,E1 -20999.415,E2 -20999.415} C_VEL
LIN {X 0,Y 223.521,Z 554.016,A -85,B 0,C 180,E1 -21000.465,E2 -21000.465} C_VEL
LIN {X 0,Y 225.406,Z 543.513,A -85,B 0,C 180,E1 -21001.484,E2 -21001.484} C_VEL
LIN {X 0,Y 226.995,Z 532.847,A -85,B 0,C 180,E1 -21002.242,E2 -21002.242} C_VEL
LIN {X 0,Y 227.998,Z 522.366,A -85,B 0,C 180,E1 -21002.781,E2 -21002.781} C_VEL
LIN {X 0,Y 229.121,Z 497.778,A -85,B 0,C 180,E1 -21003.583,E2 -21003.583} C_VEL
LIN {X 0,Y 230.096,Z 473.407,A -85,B 0,C 180,E1 -21004.319,E2 -21004.319} C_VEL
LIN {X 0,Y 226.936,Z 454.062,A -85,B 0,C 180,E1 -21005.594,E2 -21005.594} C_VEL
LIN {X 0,Y 223.215,Z 444.731,A -85,B 0,C 180,E1 -21006.64,E2 -21006.64} C_VEL
LIN {X 0,Y 217.129,Z 431.589,A -85,B 0,C 180,E1 -21008.375,E2 -21008.375} C_VEL
LIN {X 0,Y 212.237,Z 422.208,A -85,B 0,C 180,E1 -21009.824,E2 -21009.824} C_VEL
LIN {X 0,Y 210.068,Z 418.381,A -85,B 0,C 180,E1 -21010.483,E2 -21010.483} C_VEL
LIN {X 0,Y 208.181,Z 414.601,A -85,B 0,C 180,E1 -21011.18,E2 -21011.18} C_VEL
LIN {X 0,Y 207.331,Z 411.025,A -85,B 0,C 180,E1 -21013.574,E2 -21013.574} C_VEL
LIN {X 0,Y 206.775,Z 408.286,A -85,B 0,C 180,E1 -21015.715,E2 -21015.715} C_VEL
LIN {X 0,Y 206.73,Z 408.215,A -85,B 0,C 180,E1 -21019.764,E2 -21019.764} C_VEL
LIN {X 0,Y 206.729,Z 408.231,A -85,B 0,C 180,E1 -21022.269,E2 -21022.269} C_VEL
LIN {X 0,Y 206.712,Z 408.211,A -85,B 0,C 180,E1 -21027.043,E2 -21027.043} C_VEL
LIN {X 0,Y 206.769,Z 408.197,A -85,B 0,C 180,E1 -21032.096,E2 -21032.096} C_VEL
LIN {X 0,Y 206.788,Z 408.223,A -85,B 0,C 180,E1 -21036.583,E2 -21036.583} C_VEL
LIN {X 0,Y 206.875,Z 408.171,A -85,B 0,C 180,E1 -21042.196,E2 -21042.196} C_VEL
LIN {X 0,Y 206.915,Z 408.207,A -85,B 0,C 180,E1 -21046.245,E2 -21046.245} C_VEL
LIN {X 0,Y 207.107,Z 408.135,A -85,B 0,C 180,E1 -21050.23,E2 -21050.23} C_VEL
LIN {X 0,Y 207.169,Z 408.137,A -85,B 0,C 180,E1 -21052.2,E2 -21052.2} C_VEL
LIN {X 0,Y 207.383,Z 408.122,A -85,B 0,C 180,E1 -21058.057,E2 -21058.057} C_VEL
LIN {X 0,Y 207.512,Z 408.085,A -85,B 0,C 180,E1 -21059.999,E2 -21059.999} C_VEL
LIN {X 0,Y 207.383,Z 408.11,A -85,B 0,C 180,E1 -21061.941,E2 -21061.941} C_VEL
LIN {X 0,Y 207.178,Z 408.149,A -85,B 0,C 180,E1 -21067.797,E2 -21067.797} C_VEL
LIN {X 0,Y 206.981,Z 408.165,A -85,B 0,C 180,E1 -21071.754,E2 -21071.754} C_VEL
LIN {X 0,Y 206.867,Z 408.212,A -85,B 0,C 180,E1 -21075.769,E2 -21075.769} C_VEL
LIN {X 0,Y 206.782,Z 408.186,A -85,B 0,C 180,E1 -21079.868,E2 -21079.868} C_VEL
LIN {X 0,Y 206.762,Z 408.229,A -85,B 0,C 180,E1 -21084.071,E2 -21084.071} C_VEL
LIN {X 0,Y 206.735,Z 408.202,A -85,B 0,C 180,E1 -21088.419,E2 -21088.419} C_VEL
LIN {X 0,Y 206.703,Z 408.219,A -85,B 0,C 180,E1 -21092.955,E2 -21092.955} C_VEL
LIN {X 0,Y 206.72,Z 408.209,A -85,B 0,C 180,E1 -21095.319,E2 -21095.319} C_VEL
LIN {X 0,Y 206.664,Z 408.22,A -85,B 0,C 180,E1 -21100.249,E2 -21100.249} C_VEL
LIN {X 0,Y 206.634,Z 408.225,A -85,B 0,C 180,E1 -21104.418,E2 -21104.418} C_VEL
LIN {X 0,Y 206.689,Z 408.423,A -85,B 0,C 180,E1 -21108.334,E2 -21108.334} C_VEL
LIN {X 0,Y 206.921,Z 409.356,A -85,B 0,C 180,E1 -21108.718,E2 -21108.718} C_VEL
LIN {X 0,Y 208.495,Z 412.112,A -85,B 0,C 180,E1 -21109.256,E2 -21109.256} C_VEL
LIN {X 0,Y 209.582,Z 413.434,A -85,B 0,C 180,E1 -21109.572,E2 -21109.572} C_VEL
LIN {X 0,Y 218.39,Z 427.469,A -85,B 0,C 180,E1 -21112.103,E2 -21112.103} C_VEL
LIN {X 0,Y 227.159,Z 443.6,A -85,B 0,C 180,E1 -21114.435,E2 -21114.435} C_VEL
LIN {X 0,Y 235.961,Z 461.285,A -85,B 0,C 180,E1 -21116.595,E2 -21116.595} C_VEL
LIN {X 0,Y 244.153,Z 474.206,A -85,B 0,C 180,E1 -21118.302,E2 -21118.302} C_VEL
LIN {X 0,Y 252.157,Z 484.751,A -85,B 0,C 180,E1 -21119.769,E2 -21119.769} C_VEL
LIN {X 0,Y 265.439,Z 499.508,A -85,B 0,C 180,E1 -21121.884,E2 -21121.884} C_VEL
LIN {X 0,Y 276.632,Z 510.175,A -85,B 0,C 180,E1 -21123.475,E2 -21123.475} C_VEL
LIN {X 0,Y 287.008,Z 519.202,A -85,B 0,C 180,E1 -21124.959,E2 -21124.959} C_VEL
LIN {X 0,Y 298.603,Z 528.541,A -85,B 0,C 180,E1 -21126.621,E2 -21126.621} C_VEL
LIN {X 0,Y 307.018,Z 535.06,A -85,B 0,C 180,E1 -21127.984,E2 -21127.984} C_VEL
LIN {X 0,Y 315.181,Z 540.925,A -85,B 0,C 180,E1 -21129.474,E2 -21129.474} C_VEL
LIN {X 0,Y 321.84,Z 545.914,A -85,B 0,C 180,E1 -21130.879,E2 -21130.879} C_VEL
LIN {X 0,Y 329.425,Z 551.102,A -85,B 0,C 180,E1 -21132.622,E2 -21132.622} C_VEL
LIN {X 0,Y 335.758,Z 555.714,A -85,B 0,C 180,E1 -21134.333,E2 -21134.333} C_VEL
LIN {X 0,Y 340.745,Z 558.885,A -85,B 0,C 180,E1 -21135.784,E2 -21135.784} C_VEL
LIN {X 0,Y 345.69,Z 561.787,A -85,B 0,C 180,E1 -21137.381,E2 -21137.381} C_VEL
LIN {X 0,Y 350.43,Z 565.315,A -85,B 0,C 180,E1 -21139.327,E2 -21139.327} C_VEL
LIN {X 0,Y 355.186,Z 568.285,A -85,B 0,C 180,E1 -21141.622,E2 -21141.622} C_VEL
LIN {X 0,Y 357.99,Z 569.719,A -85,B 0,C 180,E1 -21143.235,E2 -21143.235} C_VEL
LIN {X 0,Y 359.998,Z 570.601,A -85,B 0,C 180,E1 -21144.638,E2 -21144.638} C_VEL
LIN {X 0,Y 362.148,Z 571.333,A -85,B 0,C 180,E1 -21146.662,E2 -21146.662} C_VEL
LIN {X 0,Y 362.833,Z 571.701,A -85,B 0,C 180,E1 -21147.78,E2 -21147.78} C_VEL
LIN {X 0,Y 363.201,Z 571.971,A -85,B 0,C 180,E1 -21148.891,E2 -21148.891} C_VEL
LIN {X 0,Y 363.421,Z 571.916,A -85,B 0,C 180,E1 -21150,E2 -21150} C_VEL
LIN {X 0,Y 363.238,Z 571.902,A -85,B 0,C 180,E1 -21151.108,E2 -21151.108} C_VEL
LIN {X 0,Y 362.834,Z 571.671,A -85,B 0,C 180,E1 -21152.22,E2 -21152.22} C_VEL
LIN {X 0,Y 362.123,Z 571.33,A -85,B 0,C 180,E1 -21153.337,E2 -21153.337} C_VEL
LIN {X 0,Y 359.986,Z 570.632,A -85,B 0,C 180,E1 -21155.341,E2 -21155.341} C_VEL
LIN {X 0,Y 357.963,Z 569.726,A -85,B 0,C 180,E1 -21156.765,E2 -21156.765} C_VEL
LIN {X 0,Y 355.194,Z 568.29,A -85,B 0,C 180,E1 -21158.387,E2 -21158.387} C_VEL
LIN {X 0,Y 350.417,Z 565.349,A -85,B 0,C 180,E1 -21160.662,E2 -21160.662} C_VEL
LIN {X 0,Y 345.683,Z 561.755,A -85,B 0,C 180,E1 -21162.614,E2 -21162.614} C_VEL
LIN {X 0,Y 340.287,Z 558.614,A -85,B 0,C 180,E1 -21164.349,E2 -21164.349} C_VEL
LIN {X 0,Y 333.105,Z 553.795,A -85,B 0,C 180,E1 -21166.407,E2 -21166.407} C_VEL
LIN {X 0,Y 327.6,Z 549.781,A -85,B 0,C 180,E1 -21167.83,E2 -21167.83} C_VEL
LIN {X 0,Y 320.442,Z 544.945,A -85,B 0,C 180,E1 -21169.426,E2 -21169.426} C_VEL
LIN {X 0,Y 312.046,Z 538.656,A -85,B 0,C 180,E1 -21171.121,E2 -21171.121} C_VEL
LIN {X 0,Y 304.258,Z 532.869,A -85,B 0,C 180,E1 -21172.491,E2 -21172.491} C_VEL
LIN {X 0,Y 296.911,Z 527.241,A -85,B 0,C 180,E1 -21173.627,E2 -21173.627} C_VEL
LIN {X 0,Y 282.28,Z 515.28,A -85,B 0,C 180,E1 -21175.717,E2 -21175.717} C_VEL
LIN {X 0,Y 269.475,Z 503.517,A -85,B 0,C 180,E1 -21177.537,E2 -21177.537} C_VEL
LIN {X 0,Y 255.834,Z 489.154,A -85,B 0,C 180,E1 -21179.609,E2 -21179.609} C_VEL
LIN {X 0,Y 246.055,Z 476.914,A -85,B 0,C 180,E1 -21181.332,E2 -21181.332} C_VEL
LIN {X 0,Y 238.134,Z 464.937,A -85,B 0,C 180,E1 -21182.93,E2 -21182.93} C_VEL
LIN {X 0,Y 231.422,Z 452.553,A -85,B 0,C 180,E1 -21184.477,E2 -21184.477} C_VEL
LIN {X 0,Y 224.525,Z 438.587,A -85,B 0,C 180,E1 -21186.246,E2 -21186.246} C_VEL
LIN {X 0,Y 216.44,Z 424.185,A -85,B 0,C 180,E1 -21188.439,E2 -21188.439} C_VEL
LIN {X 0,Y 210.657,Z 415.34,A -85,B 0,C 180,E1 -21190.094,E2 -21190.094} C_VEL
LIN {X 0,Y 208.855,Z 412.463,A -85,B 0,C 180,E1 -21190.643,E2 -21190.643} C_VEL
LIN {X 0,Y 207.205,Z 410.093,A -85,B 0,C 180,E1 -21191.153,E2 -21191.153} C_VEL
LIN {X 0,Y 206.756,Z 408.782,A -85,B 0,C 180,E1 -21191.453,E2 -21191.453} C_VEL
LIN {X 0,Y 206.62,Z 408.222,A -85,B 0,C 180,E1 -21192.133,E2 -21192.133} C_VEL
LIN {X 0,Y 206.674,Z 408.236,A -85,B 0,C 180,E1 -21197.15,E2 -21197.15} C_VEL
LIN {X 0,Y 206.713,Z 408.239,A -85,B 0,C 180,E1 -21202.269,E2 -21202.269} C_VEL
LIN {X 0,Y 206.704,Z 408.219,A -85,B 0,C 180,E1 -21207.045,E2 -21207.045} C_VEL
LIN {X 0,Y 206.762,Z 408.195,A -85,B 0,C 180,E1 -21212.097,E2 -21212.097} C_VEL
LIN {X 0,Y 206.781,Z 408.229,A -85,B 0,C 180,E1 -21216.584,E2 -21216.584} C_VEL
LIN {X 0,Y 206.868,Z 408.181,A -85,B 0,C 180,E1 -21222.197,E2 -21222.197} C_VEL
LIN {X 0,Y 206.91,Z 408.206,A -85,B 0,C 180,E1 -21226.246,E2 -21226.246} C_VEL
LIN {X 0,Y 207.101,Z 408.139,A -85,B 0,C 180,E1 -21230.232,E2 -21230.232} C_VEL
LIN {X 0,Y 207.174,Z 408.15,A -85,B 0,C 180,E1 -21232.202,E2 -21232.202} C_VEL
LIN {X 0,Y 207.379,Z 408.111,A -85,B 0,C 180,E1 -21238.059,E2 -21238.059} C_VEL
LIN {X 0,Y 207.508,Z 408.086,A -85,B 0,C 180,E1 -21240.001,E2 -21240.001} C_VEL
LIN {X 0,Y 207.379,Z 408.122,A -85,B 0,C 180,E1 -21241.943,E2 -21241.943} C_VEL
LIN {X 0,Y 207.165,Z 408.138,A -85,B 0,C 180,E1 -21247.8,E2 -21247.8} C_VEL
LIN {X 0,Y 206.979,Z 408.173,A -85,B 0,C 180,E1 -21251.756,E2 -21251.756} C_VEL
LIN {X 0,Y 206.865,Z 408.199,A -85,B 0,C 180,E1 -21255.772,E2 -21255.772} C_VEL
LIN {X 0,Y 206.781,Z 408.188,A -85,B 0,C 180,E1 -21259.87,E2 -21259.87} C_VEL
LIN {X 0,Y 206.762,Z 408.219,A -85,B 0,C 180,E1 -21264.073,E2 -21264.073} C_VEL
LIN {X 0,Y 206.743,Z 408.206,A -85,B 0,C 180,E1 -21268.42,E2 -21268.42} C_VEL
LIN {X 0,Y 206.708,Z 408.211,A -85,B 0,C 180,E1 -21272.957,E2 -21272.957} C_VEL
LIN {X 0,Y 206.725,Z 408.232,A -85,B 0,C 180,E1 -21277.731,E2 -21277.731} C_VEL
LIN {X 0,Y 206.726,Z 408.228,A -85,B 0,C 180,E1 -21281.591,E2 -21281.591} C_VEL
LIN {X 0,Y 206.766,Z 408.416,A -85,B 0,C 180,E1 -21284.457,E2 -21284.457} C_VEL
LIN {X 0,Y 208.119,Z 414.359,A -85,B 0,C 180,E1 -21288.718,E2 -21288.718} C_VEL
LIN {X 0,Y 208.804,Z 416.244,A -85,B 0,C 180,E1 -21289.122,E2 -21289.122} C_VEL
LIN {X 0,Y 211.489,Z 420.802,A -85,B 0,C 180,E1 -21289.947,E2 -21289.947} C_VEL
LIN {X 0,Y 215.932,Z 429.135,A -85,B 0,C 180,E1 -21291.273,E2 -21291.273} C_VEL
LIN {X 0,Y 222.987,Z 444.148,A -85,B 0,C 180,E1 -21293.294,E2 -21293.294} C_VEL
LIN {X 0,Y 226.885,Z 453.934,A -85,B 0,C 180,E1 -21294.392,E2 -21294.392} C_VEL
LIN {X 0,Y 230.128,Z 473.73,A -85,B 0,C 180,E1 -21295.698,E2 -21295.698} C_VEL
LIN {X 0,Y 228.013,Z 521.322,A -85,B 0,C 180,E1 -21297.166,E2 -21297.166} C_VEL
LIN {X 0,Y 227.111,Z 531.431,A -85,B 0,C 180,E1 -21297.669,E2 -21297.669} C_VEL
LIN {X 0,Y 225.802,Z 541.002,A -85,B 0,C 180,E1 -21298.318,E2 -21298.318} C_VEL
LIN {X 0,Y 224.309,Z 550.092,A -85,B 0,C 180,E1 -21299.133,E2 -21299.133} C_VEL
LIN {X 0,Y 222.477,Z 559.234,A -85,B 0,C 180,E1 -21300.164,E2 -21300.164} C_VEL
LIN {X 0,Y 221.506,Z 563.832,A -85,B 0,C 180,E1 -21300.775,E2 -21300.775} C_VEL
LIN {X 0,Y 219.805,Z 568.882,A -85,B 0,C 180,E1 -21301.434,E2 -21301.434} C_VEL
LIN {X 0,Y 215.141,Z 576.697,A -85,B 0,C 180,E1 -21302.471,E2 -21302.471} C_VEL
LIN {X 0,Y 210.31,Z 584.189,A -85,B 0,C 180,E1 -21303.708,E2 -21303.708} C_VEL
LIN {X 0,Y 208.363,Z 588.38,A -85,B 0,C 180,E1 -21304.676,E2 -21304.676} C_VEL
LIN {X 0,Y 205.608,Z 597.219,A -85,B 0,C 180,E1 -21307.24,E2 -21307.24} C_VEL
LIN {X 0,Y 202.923,Z 605.272,A -85,B 0,C 180,E1 -21310.265,E2 -21310.265} C_VEL
LIN {X 0,Y 201.145,Z 610.546,A -85,B 0,C 180,E1 -21312.724,E2 -21312.724} C_VEL
LIN {X 0,Y 199.388,Z 615.639,A -85,B 0,C 180,E1 -21315.716,E2 -21315.716} C_VEL
LIN {X 0,Y 198.272,Z 619.609,A -85,B 0,C 180,E1 -21318.759,E2 -21318.759} C_VEL
LIN {X 0,Y 197.591,Z 622.549,A -85,B 0,C 180,E1 -21321.821,E2 -21321.821} C_VEL
LIN {X 0,Y 197.343,Z 624.054,A -85,B 0,C 180,E1 -21323.868,E2 -21323.868} C_VEL
LIN {X 0,Y 197.241,Z 625.586,A -85,B 0,C 180,E1 -21327.959,E2 -21327.959} C_VEL
LIN {X 0,Y 197.339,Z 625.869,A -85,B 0,C 180,E1 -21330.001,E2 -21330.001} C_VEL
LIN {X 0,Y 197.21,Z 624.985,A -85,B 0,C 180,E1 -21334.088,E2 -21334.088} C_VEL
LIN {X 0,Y 197.314,Z 624.053,A -85,B 0,C 180,E1 -21336.135,E2 -21336.135} C_VEL
LIN {X 0,Y 198.022,Z 620.699,A -85,B 0,C 180,E1 -21340.222,E2 -21340.222} C_VEL
LIN {X 0,Y 198.997,Z 617.068,A -85,B 0,C 180,E1 -21343.272,E2 -21343.272} C_VEL
LIN {X 0,Y 200.502,Z 612.334,A -85,B 0,C 180,E1 -21346.285,E2 -21346.285} C_VEL
LIN {X 0,Y 202.534,Z 606.362,A -85,B 0,C 180,E1 -21349.248,E2 -21349.248} C_VEL
LIN {X 0,Y 204.688,Z 600.273,A -85,B 0,C 180,E1 -21351.661,E2 -21351.661} C_VEL
LIN {X 0,Y 206.385,Z 594.683,A -85,B 0,C 180,E1 -21353.533,E2 -21353.533} C_VEL
LIN {X 0,Y 208.546,Z 587.872,A -85,B 0,C 180,E1 -21355.447,E2 -21355.447} C_VEL
LIN {X 0,Y 210.959,Z 580.049,A -85,B 0,C 180,E1 -21357.263,E2 -21357.263} C_VEL
LIN {X 0,Y 213.195,Z 571.968,A -85,B 0,C 180,E1 -21358.824,E2 -21358.824} C_VEL
LIN {X 0,Y 215.652,Z 562.211,A -85,B 0,C 180,E1 -21360.341,E2 -21360.341} C_VEL
LIN {X 0,Y 217.446,Z 553.822,A -85,B 0,C 180,E1 -21361.411,E2 -21361.411} C_VEL
LIN {X 0,Y 219.396,Z 543.319,A -85,B 0,C 180,E1 -21362.45,E2 -21362.45} C_VEL
LIN {X 0,Y 220.885,Z 533.527,A -85,B 0,C 180,E1 -21363.178,E2 -21363.178} C_VEL
LIN {X 0,Y 222.025,Z 522.885,A -85,B 0,C 180,E1 -21363.743,E2 -21363.743} C_VEL
LIN {X 0,Y 223.022,Z 502.755,A -85,B 0,C 180,E1 -21364.432,E2 -21364.432} C_VEL
LIN {X 0,Y 224.199,Z 474.298,A -85,B 0,C 180,E1 -21365.312,E2 -21365.312} C_VEL
LIN {X 0,Y 221.239,Z 456.03,A -85,B 0,C 180,E1 -21366.571,E2 -21366.571} C_VEL
LIN {X 0,Y 214.262,Z 439.7,A -85,B 0,C 180,E1 -21368.64,E2 -21368.64} C_VEL
LIN {X 0,Y 208.217,Z 427.589,A -85,B 0,C 180,E1 -21370.507,E2 -21370.507} C_VEL
LIN {X 0,Y 205.167,Z 422.321,A -85,B 0,C 180,E1 -21371.474,E2 -21371.474} C_VEL
LIN {X 0,Y 202.893,Z 418.28,A -85,B 0,C 180,E1 -21372.228,E2 -21372.228} C_VEL
LIN {X 0,Y 200.891,Z 414.357,A -85,B 0,C 180,E1 -21373.023,E2 -21373.023} C_VEL
LIN {X 0,Y 200.139,Z 411.002,A -85,B 0,C 180,E1 -21375.386,E2 -21375.386} C_VEL
LIN {X 0,Y 199.696,Z 409.155,A -85,B 0,C 180,E1 -21377.039,E2 -21377.039} C_VEL
LIN {X 0,Y 199.684,Z 409.093,A -85,B 0,C 180,E1 -21380.742,E2 -21380.742} C_VEL
LIN {X 0,Y 199.637,Z 409.088,A -85,B 0,C 180,E1 -21385.717,E2 -21385.717} C_VEL
LIN {X 0,Y 199.707,Z 409.095,A -85,B 0,C 180,E1 -21388.137,E2 -21388.137} C_VEL
LIN {X 0,Y 199.689,Z 409.073,A -85,B 0,C 180,E1 -21392.771,E2 -21392.771} C_VEL
LIN {X 0,Y 199.74,Z 409.102,A -85,B 0,C 180,E1 -21397.228,E2 -21397.228} C_VEL
LIN {X 0,Y 199.798,Z 409.05,A -85,B 0,C 180,E1 -21401.757,E2 -21401.757} C_VEL
LIN {X 0,Y 199.85,Z 409.088,A -85,B 0,C 180,E1 -21405.748,E2 -21405.748} C_VEL
LIN {X 0,Y 200.072,Z 409.012,A -85,B 0,C 180,E1 -21409.883,E2 -21409.883} C_VEL
LIN {X 0,Y 200.036,Z 409.056,A -85,B 0,C 180,E1 -21413.949,E2 -21413.949} C_VEL
LIN {X 0,Y 200.323,Z 409.001,A -85,B 0,C 180,E1 -21417.988,E2 -21417.988} C_VEL
LIN {X 0,Y 200.476,Z 408.961,A -85,B 0,C 180,E1 -21419.999,E2 -21419.999} C_VEL
LIN {X 0,Y 200.032,Z 409.06,A -85,B 0,C 180,E1 -21424.028,E2 -21424.028} C_VEL
LIN {X 0,Y 200.119,Z 409.022,A -85,B 0,C 180,E1 -21428.074,E2 -21428.074} C_VEL
LIN {X 0,Y 199.914,Z 409.05,A -85,B 0,C 180,E1 -21432.176,E2 -21432.176} C_VEL
LIN {X 0,Y 199.805,Z 409.082,A -85,B 0,C 180,E1 -21436.342,E2 -21436.342} C_VEL
LIN {X 0,Y 199.699,Z 409.073,A -85,B 0,C 180,E1 -21440.604,E2 -21440.604} C_VEL
LIN {X 0,Y 199.671,Z 409.099,A -85,B 0,C 180,E1 -21444.983,E2 -21444.983} C_VEL
LIN {X 0,Y 199.663,Z 409.095,A -85,B 0,C 180,E1 -21449.523,E2 -21449.523} C_VEL
LIN {X 0,Y 199.656,Z 409.105,A -85,B 0,C 180,E1 -21452.348,E2 -21452.348} C_VEL
LIN {X 0,Y 199.638,Z 409.106,A -85,B 0,C 180,E1 -21456.758,E2 -21456.758} C_VEL
LIN {X 0,Y 199.637,Z 409.102,A -85,B 0,C 180,E1 -21459.32,E2 -21459.32} C_VEL
LIN {X 0,Y 199.58,Z 409.092,A -85,B 0,C 180,E1 -21464.77,E2 -21464.77} C_VEL
LIN {X 0,Y 199.626,Z 409.449,A -85,B 0,C 180,E1 -21466.633,E2 -21466.633} C_VEL
LIN {X 0,Y 200.034,Z 410.814,A -85,B 0,C 180,E1 -21467.045,E2 -21467.045} C_VEL
LIN {X 0,Y 201.781,Z 413.406,A -85,B 0,C 180,E1 -21467.643,E2 -21467.643} C_VEL
LIN {X 0,Y 202.817,Z 414.721,A -85,B 0,C 180,E1 -21467.972,E2 -21467.972} C_VEL
LIN {X 0,Y 205.033,Z 417.96,A -85,B 0,C 180,E1 -21468.68,E2 -21468.68} C_VEL
LIN {X 0,Y 213.822,Z 432.072,A -85,B 0,C 180,E1 -21471.332,E2 -21471.332} C_VEL
LIN {X 0,Y 222.007,Z 447.336,A -85,B 0,C 180,E1 -21473.619,E2 -21473.619} C_VEL
LIN {X 0,Y 231.117,Z 465.783,A -85,B 0,C 180,E1 -21475.959,E2 -21475.959} C_VEL
LIN {X 0,Y 239.035,Z 478.416,A -85,B 0,C 180,E1 -21477.683,E2 -21477.683} C_VEL
LIN {X 0,Y 247.444,Z 489.639,A -85,B 0,C 180,E1 -21479.288,E2 -21479.288} C_VEL
LIN {X 0,Y 260.707,Z 504.497,A -85,B 0,C 180,E1 -21481.477,E2 -21481.477} C_VEL
LIN {X 0,Y 271.865,Z 515.352,A -85,B 0,C 180,E1 -21483.208,E2 -21483.208} C_VEL
LIN {X 0,Y 282.944,Z 525.028,A -85,B 0,C 180,E1 -21484.936,E2 -21484.936} C_VEL
LIN {X 0,Y 295.738,Z 535.222,A -85,B 0,C 180,E1 -21486.898,E2 -21486.898} C_VEL
LIN {X 0,Y 304.259,Z 541.804,A -85,B 0,C 180,E1 -21488.31,E2 -21488.31} C_VEL
LIN {X 0,Y 310.773,Z 546.453,A -85,B 0,C 180,E1 -21489.515,E2 -21489.515} C_VEL
LIN {X 0,Y 316.461,Z 550.779,A -85,B 0,C 180,E1 -21490.703,E2 -21490.703} C_VEL
LIN {X 0,Y 324.309,Z 556.13,A -85,B 0,C 180,E1 -21492.458,E2 -21492.458} C_VEL
LIN {X 0,Y 329.845,Z 560.219,A -85,B 0,C 180,E1 -21493.919,E2 -21493.919} C_VEL
LIN {X 0,Y 335.132,Z 563.724,A -85,B 0,C 180,E1 -21495.425,E2 -21495.425} C_VEL
LIN {X 0,Y 341.104,Z 567.247,A -85,B 0,C 180,E1 -21497.308,E2 -21497.308} C_VEL
LIN {X 0,Y 344.2,Z 569.567,A -85,B 0,C 180,E1 -21498.541,E2 -21498.541} C_VEL
LIN {X 0,Y 346.373,Z 571.14,A -85,B 0,C 180,E1 -21499.478,E2 -21499.478} C_VEL
LIN {X 0,Y 349.089,Z 572.864,A -85,B 0,C 180,E1 -21500.731,E2 -21500.731} C_VEL
LIN {X 0,Y 351.448,Z 574.232,A -85,B 0,C 180,E1 -21501.953,E2 -21501.953} C_VEL
LIN {X 0,Y 353.802,Z 575.405,A -85,B 0,C 180,E1 -21503.313,E2 -21503.313} C_VEL
LIN {X 0,Y 355.28,Z 576.088,A -85,B 0,C 180,E1 -21504.323,E2 -21504.323} C_VEL
LIN {X 0,Y 356.699,Z 576.69,A -85,B 0,C 180,E1 -21505.479,E2 -21505.479} C_VEL
LIN {X 0,Y 357.867,Z 577.007,A -85,B 0,C 180,E1 -21506.622,E2 -21506.622} C_VEL
LIN {X 0,Y 358.662,Z 577.429,A -85,B 0,C 180,E1 -21507.908,E2 -21507.908} C_VEL
LIN {X 0,Y 359.181,Z 577.586,A -85,B 0,C 180,E1 -21510,E2 -21510} C_VEL
LIN {X 0,Y 358.655,Z 577.408,A -85,B 0,C 180,E1 -21512.063,E2 -21512.063} C_VEL
LIN {X 0,Y 357.836,Z 577.006,A -85,B 0,C 180,E1 -21513.377,E2 -21513.377} C_VEL
LIN {X 0,Y 356.671,Z 576.678,A -85,B 0,C 180,E1 -21514.52,E2 -21514.52} C_VEL
LIN {X 0,Y 355.238,Z 576.092,A -85,B 0,C 180,E1 -21515.677,E2 -21515.677} C_VEL
LIN {X 0,Y 353.478,Z 575.289,A -85,B 0,C 180,E1 -21516.851,E2 -21516.851} C_VEL
LIN {X 0,Y 351.435,Z 574.219,A -85,B 0,C 180,E1 -21518.047,E2 -21518.047} C_VEL
LIN {X 0,Y 348.972,Z 572.792,A -85,B 0,C 180,E1 -21519.318,E2 -21519.318} C_VEL
LIN {X 0,Y 346.341,Z 571.147,A -85,B 0,C 180,E1 -21520.522,E2 -21520.522} C_VEL
LIN {X 0,Y 342.275,Z 568.099,A -85,B 0,C 180,E1 -21522.251,E2 -21522.251} C_VEL
LIN {X 0,Y 337.75,Z 565.291,A -85,B 0,C 180,E1 -21523.772,E2 -21523.772} C_VEL
LIN {X 0,Y 331.707,Z 561.464,A -85,B 0,C 180,E1 -21525.566,E2 -21525.566} C_VEL
LIN {X 0,Y 325.913,Z 557.313,A -85,B 0,C 180,E1 -21527.138,E2 -21527.138} C_VEL
LIN {X 0,Y 319.104,Z 552.65,A -85,B 0,C 180,E1 -21528.734,E2 -21528.734} C_VEL
LIN {X 0,Y 312.293,Z 547.715,A -85,B 0,C 180,E1 -21530.178,E2 -21530.178} C_VEL
LIN {X 0,Y 305.751,Z 542.901,A -85,B 0,C 180,E1 -21531.424,E2 -21531.424} C_VEL
LIN {X 0,Y 297.411,Z 536.519,A -85,B 0,C 180,E1 -21532.842,E2 -21532.842} C_VEL
LIN {X 0,Y 284.429,Z 526.271,A -85,B 0,C 180,E1 -21534.837,E2 -21534.837} C_VEL
LIN {X 0,Y 273.823,Z 517.137,A -85,B 0,C 180,E1 -21536.48,E2 -21536.48} C_VEL
LIN {X 0,Y 263.773,Z 507.562,A -85,B 0,C 180,E1 -21538.046,E2 -21538.046} C_VEL
LIN {X 0,Y 250.928,Z 493.843,A -85,B 0,C 180,E1 -21540.1,E2 -21540.1} C_VEL
LIN {X 0,Y 241.326,Z 481.705,A -85,B 0,C 180,E1 -21541.858,E2 -21541.858} C_VEL
LIN {X 0,Y 233.36,Z 469.606,A -85,B 0,C 180,E1 -21543.528,E2 -21543.528} C_VEL
LIN {X 0,Y 226.365,Z 456.577,A -85,B 0,C 180,E1 -21545.214,E2 -21545.214} C_VEL
LIN {X 0,Y 219.55,Z 442.613,A -85,B 0,C 180,E1 -21547.048,E2 -21547.048} C_VEL
LIN {X 0,Y 211.69,Z 428.467,A -85,B 0,C 180,E1 -21549.29,E2 -21549.29} C_VEL
LIN {X 0,Y 204.604,Z 417.49,A -85,B 0,C 180,E1 -21551.448,E2 -21551.448} C_VEL
LIN {X 0,Y 201.957,Z 413.567,A -85,B 0,C 180,E1 -21552.304,E2 -21552.304} C_VEL
LIN {X 0,Y 200.152,Z 411.042,A -85,B 0,C 180,E1 -21552.907,E2 -21552.907} C_VEL
LIN {X 0,Y 199.638,Z 409.518,A -85,B 0,C 180,E1 -21553.325,E2 -21553.325} C_VEL
LIN {X 0,Y 199.597,Z 409.199,A -85,B 0,C 180,E1 -21553.64,E2 -21553.64} C_VEL
LIN {X 0,Y 199.624,Z 409.102,A -85,B 0,C 180,E1 -21558.018,E2 -21558.018} C_VEL
LIN {X 0,Y 199.639,Z 409.102,A -85,B 0,C 180,E1 -21560.756,E2 -21560.756} C_VEL
LIN {X 0,Y 199.629,Z 409.09,A -85,B 0,C 180,E1 -21565.718,E2 -21565.718} C_VEL
LIN {X 0,Y 199.699,Z 409.108,A -85,B 0,C 180,E1 -21568.138,E2 -21568.138} C_VEL
LIN {X 0,Y 199.681,Z 409.076,A -85,B 0,C 180,E1 -21572.772,E2 -21572.772} C_VEL
LIN {X 0,Y 199.733,Z 409.103,A -85,B 0,C 180,E1 -21577.23,E2 -21577.23} C_VEL
LIN {X 0,Y 199.792,Z 409.058,A -85,B 0,C 180,E1 -21581.759,E2 -21581.759} C_VEL
LIN {X 0,Y 199.844,Z 409.091,A -85,B 0,C 180,E1 -21585.75,E2 -21585.75} C_VEL
LIN {X 0,Y 200.066,Z 409.014,A -85,B 0,C 180,E1 -21589.885,E2 -21589.885} C_VEL
LIN {X 0,Y 200.035,Z 409.065,A -85,B 0,C 180,E1 -21593.951,E2 -21593.951} C_VEL
LIN {X 0,Y 200.319,Z 408.99,A -85,B 0,C 180,E1 -21597.991,E2 -21597.991} C_VEL
LIN {X 0,Y 200.473,Z 408.961,A -85,B 0,C 180,E1 -21600.001,E2 -21600.001} C_VEL
LIN {X 0,Y 200.03,Z 409.067,A -85,B 0,C 180,E1 -21604.031,E2 -21604.031} C_VEL
LIN {X 0,Y 200.109,Z 409.013,A -85,B 0,C 180,E1 -21608.077,E2 -21608.077} C_VEL
LIN {X 0,Y 199.911,Z 409.06,A -85,B 0,C 180,E1 -21612.178,E2 -21612.178} C_VEL
LIN {X 0,Y 199.802,Z 409.066,A -85,B 0,C 180,E1 -21616.345,E2 -21616.345} C_VEL
LIN {X 0,Y 199.698,Z 409.079,A -85,B 0,C 180,E1 -21620.607,E2 -21620.607} C_VEL
LIN {X 0,Y 199.671,Z 409.085,A -85,B 0,C 180,E1 -21624.986,E2 -21624.986} C_VEL
LIN {X 0,Y 199.674,Z 409.103,A -85,B 0,C 180,E1 -21629.524,E2 -21629.524} C_VEL
LIN {X 0,Y 199.663,Z 409.094,A -85,B 0,C 180,E1 -21632.353,E2 -21632.353} C_VEL
LIN {X 0,Y 199.653,Z 409.114,A -85,B 0,C 180,E1 -21636.758,E2 -21636.758} C_VEL
LIN {X 0,Y 199.679,Z 409.094,A -85,B 0,C 180,E1 -21639.313,E2 -21639.313} C_VEL
LIN {X 0,Y 199.715,Z 409.192,A -85,B 0,C 180,E1 -21643.115,E2 -21643.115} C_VEL
LIN {X 0,Y 200.812,Z 414.069,A -85,B 0,C 180,E1 -21646.848,E2 -21646.848} C_VEL
LIN {X 0,Y 201.443,Z 415.793,A -85,B 0,C 180,E1 -21647.269,E2 -21647.269} C_VEL
LIN {X 0,Y 204.122,Z 420.353,A -85,B 0,C 180,E1 -21648.178,E2 -21648.178} C_VEL
LIN {X 0,Y 207.627,Z 426.59,A -85,B 0,C 180,E1 -21649.31,E2 -21649.31} C_VEL
LIN {X 0,Y 212.933,Z 436.91,A -85,B 0,C 180,E1 -21650.958,E2 -21650.958} C_VEL
LIN {X 0,Y 219.903,Z 452.61,A -85,B 0,C 180,E1 -21653.035,E2 -21653.035} C_VEL
LIN {X 0,Y 221.499,Z 457.312,A -85,B 0,C 180,E1 -21653.529,E2 -21653.529} C_VEL
LIN {X 0,Y 224.257,Z 475.429,A -85,B 0,C 180,E1 -21654.742,E2 -21654.742} C_VEL
LIN {X 0,Y 222.123,Z 520.822,A -85,B 0,C 180,E1 -21656.163,E2 -21656.163} C_VEL
LIN {X 0,Y 221.114,Z 531.462,A -85,B 0,C 180,E1 -21656.698,E2 -21656.698} C_VEL
LIN {X 0,Y 219.802,Z 540.807,A -85,B 0,C 180,E1 -21657.347,E2 -21657.347} C_VEL
LIN {X 0,Y 218.243,Z 549.897,A -85,B 0,C 180,E1 -21658.177,E2 -21658.177} C_VEL
LIN {X 0,Y 216.323,Z 559.038,A -85,B 0,C 180,E1 -21659.224,E2 -21659.224} C_VEL
LIN {X 0,Y 214.2,Z 568.036,A -85,B 0,C 180,E1 -21660.519,E2 -21660.519} C_VEL
LIN {X 0,Y 211.838,Z 576.758,A -85,B 0,C 180,E1 -21662.057,E2 -21662.057} C_VEL
LIN {X 0,Y 209.685,Z 584.177,A -85,B 0,C 180,E1 -21663.635,E2 -21663.635} C_VEL
LIN {X 0,Y 208.363,Z 588.38,A -85,B 0,C 180,E1 -21664.676,E2 -21664.676} C_VEL
LIN {X 0,Y 206.463,Z 592.527,A -85,B 0,C 180,E1 -21665.718,E2 -21665.718} C_VEL
LIN {X 0,Y 201.732,Z 598.773,A -85,B 0,C 180,E1 -21667.431,E2 -21667.431} C_VEL
LIN {X 0,Y 197.088,Z 604.508,A -85,B 0,C 180,E1 -21669.363,E2 -21669.363} C_VEL
LIN {X 0,Y 195.356,Z 607.59,A -85,B 0,C 180,E1 -21670.728,E2 -21670.728} C_VEL
LIN {X 0,Y 193.042,Z 613.929,A -85,B 0,C 180,E1 -21674.155,E2 -21674.155} C_VEL
LIN {X 0,Y 191.65,Z 618.287,A -85,B 0,C 180,E1 -21677.29,E2 -21677.29} C_VEL
LIN {X 0,Y 190.54,Z 622.354,A -85,B 0,C 180,E1 -21681.516,E2 -21681.516} C_VEL
LIN {X 0,Y 190.281,Z 623.859,A -85,B 0,C 180,E1 -21683.639,E2 -21683.639} C_VEL
LIN {X 0,Y 190.154,Z 625.028,A -85,B 0,C 180,E1 -21686.31,E2 -21686.31} C_VEL
LIN {X 0,Y 190.243,Z 625.674,A -85,B 0,C 180,E1 -21690.001,E2 -21690.001} C_VEL
LIN {X 0,Y 190.131,Z 624.79,A -85,B 0,C 180,E1 -21694.24,E2 -21694.24} C_VEL
LIN {X 0,Y 190.234,Z 623.857,A -85,B 0,C 180,E1 -21696.364,E2 -21696.364} C_VEL
LIN {X 0,Y 191.011,Z 620.503,A -85,B 0,C 180,E1 -21700.602,E2 -21700.602} C_VEL
LIN {X 0,Y 192.044,Z 616.871,A -85,B 0,C 180,E1 -21703.761,E2 -21703.761} C_VEL
LIN {X 0,Y 193.659,Z 612.137,A -85,B 0,C 180,E1 -21706.878,E2 -21706.878} C_VEL
LIN {X 0,Y 195.809,Z 606.166,A -85,B 0,C 180,E1 -21709.937,E2 -21709.937} C_VEL
LIN {X 0,Y 197.594,Z 601.444,A -85,B 0,C 180,E1 -21711.906,E2 -21711.906} C_VEL
LIN {X 0,Y 199.319,Z 596.205,A -85,B 0,C 180,E1 -21713.812,E2 -21713.812} C_VEL
LIN {X 0,Y 202.136,Z 587.676,A -85,B 0,C 180,E1 -21716.315,E2 -21716.315} C_VEL
LIN {X 0,Y 204.649,Z 579.853,A -85,B 0,C 180,E1 -21718.177,E2 -21718.177} C_VEL
LIN {X 0,Y 206.997,Z 571.772,A -85,B 0,C 180,E1 -21719.772,E2 -21719.772} C_VEL
LIN {X 0,Y 209.55,Z 562.016,A -85,B 0,C 180,E1 -21721.322,E2 -21721.322} C_VEL
LIN {X 0,Y 211.408,Z 553.626,A -85,B 0,C 180,E1 -21722.416,E2 -21722.416} C_VEL
LIN {X 0,Y 213.455,Z 543.124,A -85,B 0,C 180,E1 -21723.47,E2 -21723.47} C_VEL
LIN {X 0,Y 215.055,Z 532.842,A -85,B 0,C 180,E1 -21724.24,E2 -21724.24} C_VEL
LIN {X 0,Y 216.18,Z 522.405,A -85,B 0,C 180,E1 -21724.799,E2 -21724.799} C_VEL
LIN {X 0,Y 217.322,Z 500.113,A -85,B 0,C 180,E1 -21725.566,E2 -21725.566} C_VEL
LIN {X 0,Y 218.401,Z 475.497,A -85,B 0,C 180,E1 -21726.341,E2 -21726.341} C_VEL
LIN {X 0,Y 215.771,Z 458.808,A -85,B 0,C 180,E1 -21727.535,E2 -21727.535} C_VEL
LIN {X 0,Y 209.172,Z 443.216,A -85,B 0,C 180,E1 -21729.602,E2 -21729.602} C_VEL
LIN {X 0,Y 203.7,Z 432.085,A -85,B 0,C 180,E1 -21731.387,E2 -21731.387} C_VEL
LIN {X 0,Y 198.038,Z 422.117,A -85,B 0,C 180,E1 -21733.321,E2 -21733.321} C_VEL
LIN {X 0,Y 195.821,Z 418.213,A -85,B 0,C 180,E1 -21734.126,E2 -21734.126} C_VEL
LIN {X 0,Y 193.674,Z 414.111,A -85,B 0,C 180,E1 -21735.049,E2 -21735.049} C_VEL
LIN {X 0,Y 193.08,Z 411.794,A -85,B 0,C 180,E1 -21736.718,E2 -21736.718} C_VEL
LIN {X 0,Y 192.629,Z 410.056,A -85,B 0,C 180,E1 -21738.367,E2 -21738.367} C_VEL
LIN {X 0,Y 192.622,Z 409.986,A -85,B 0,C 180,E1 -21743.388,E2 -21743.388} C_VEL
LIN {X 0,Y 192.61,Z 409.966,A -85,B 0,C 180,E1 -21747.059,E2 -21747.059} C_VEL
LIN {X 0,Y 192.667,Z 409.955,A -85,B 0,C 180,E1 -21751.691,E2 -21751.691} C_VEL
LIN {X 0,Y 192.708,Z 409.973,A -85,B 0,C 180,E1 -21756.348,E2 -21756.348} C_VEL
LIN {X 0,Y 192.734,Z 409.929,A -85,B 0,C 180,E1 -21761.457,E2 -21761.457} C_VEL
LIN {X 0,Y 192.774,Z 409.966,A -85,B 0,C 180,E1 -21765.213,E2 -21765.213} C_VEL
LIN {X 0,Y 192.983,Z 409.896,A -85,B 0,C 180,E1 -21769.507,E2 -21769.507} C_VEL
LIN {X 0,Y 193.063,Z 409.886,A -85,B 0,C 180,E1 -21771.626,E2 -21771.626} C_VEL
LIN {X 0,Y 193.265,Z 409.88,A -85,B 0,C 180,E1 -21777.915,E2 -21777.915} C_VEL
LIN {X 0,Y 193.441,Z 409.836,A -85,B 0,C 180,E1 -21779.999,E2 -21779.999} C_VEL
LIN {X 0,Y 192.979,Z 409.94,A -85,B 0,C 180,E1 -21784.176,E2 -21784.176} C_VEL
LIN {X 0,Y 193.068,Z 409.895,A -85,B 0,C 180,E1 -21788.371,E2 -21788.371} C_VEL
LIN {X 0,Y 192.853,Z 409.936,A -85,B 0,C 180,E1 -21792.629,E2 -21792.629} C_VEL
LIN {X 0,Y 192.757,Z 409.948,A -85,B 0,C 180,E1 -21796.957,E2 -21796.957} C_VEL
LIN {X 0,Y 192.635,Z 409.962,A -85,B 0,C 180,E1 -21801.396,E2 -21801.396} C_VEL
LIN {X 0,Y 192.663,Z 409.983,A -85,B 0,C 180,E1 -21804.223,E2 -21804.223} C_VEL
LIN {X 0,Y 192.643,Z 409.96,A -85,B 0,C 180,E1 -21808.888,E2 -21808.888} C_VEL
LIN {X 0,Y 192.596,Z 409.972,A -85,B 0,C 180,E1 -21813.185,E2 -21813.185} C_VEL
LIN {X 0,Y 192.572,Z 409.995,A -85,B 0,C 180,E1 -21818.345,E2 -21818.345} C_VEL
LIN {X 0,Y 192.512,Z 410.002,A -85,B 0,C 180,E1 -21823.102,E2 -21823.102} C_VEL
LIN {X 0,Y 192.585,Z 410.272,A -85,B 0,C 180,E1 -21824.641,E2 -21824.641} C_VEL
LIN {X 0,Y 192.902,Z 411.428,A -85,B 0,C 180,E1 -21825.05,E2 -21825.05} C_VEL
LIN {X 0,Y 194.506,Z 414.1,A -85,B 0,C 180,E1 -21825.678,E2 -21825.678} C_VEL
LIN {X 0,Y 195.789,Z 415.546,A -85,B 0,C 180,E1 -21826.119,E2 -21826.119} C_VEL
LIN {X 0,Y 198.111,Z 418.961,A -85,B 0,C 180,E1 -21826.932,E2 -21826.932} C_VEL
LIN {X 0,Y 204.317,Z 428.509,A -85,B 0,C 180,E1 -21828.987,E2 -21828.987} C_VEL
LIN {X 0,Y 210.21,Z 438.318,A -85,B 0,C 180,E1 -21830.805,E2 -21830.805} C_VEL
LIN {X 0,Y 217.857,Z 453.058,A -85,B 0,C 180,E1 -21833.037,E2 -21833.037} C_VEL
LIN {X 0,Y 226.233,Z 470.162,A -85,B 0,C 180,E1 -21835.279,E2 -21835.279} C_VEL
LIN {X 0,Y 234.324,Z 483.184,A -85,B 0,C 180,E1 -21837.116,E2 -21837.116} C_VEL
LIN {X 0,Y 242.729,Z 494.498,A -85,B 0,C 180,E1 -21838.784,E2 -21838.784} C_VEL
LIN {X 0,Y 255.555,Z 509.079,A -85,B 0,C 180,E1 -21841.028,E2 -21841.028} C_VEL
LIN {X 0,Y 265.94,Z 519.503,A -85,B 0,C 180,E1 -21842.8,E2 -21842.8} C_VEL
LIN {X 0,Y 277.688,Z 529.933,A -85,B 0,C 180,E1 -21844.793,E2 -21844.793} C_VEL
LIN {X 0,Y 290.376,Z 540.012,A -85,B 0,C 180,E1 -21846.882,E2 -21846.882} C_VEL
LIN {X 0,Y 300.185,Z 547.549,A -85,B 0,C 180,E1 -21848.532,E2 -21848.532} C_VEL
LIN {X 0,Y 307.958,Z 553.226,A -85,B 0,C 180,E1 -21849.982,E2 -21849.982} C_VEL
LIN {X 0,Y 316.95,Z 559.636,A -85,B 0,C 180,E1 -21851.914,E2 -21851.914} C_VEL
LIN {X 0,Y 323.743,Z 564.502,A -85,B 0,C 180,E1 -21853.608,E2 -21853.608} C_VEL
LIN {X 0,Y 329.29,Z 568.313,A -85,B 0,C 180,E1 -21855.16,E2 -21855.16} C_VEL
LIN {X 0,Y 334.137,Z 571.229,A -85,B 0,C 180,E1 -21856.622,E2 -21856.622} C_VEL
LIN {X 0,Y 338.08,Z 573.814,A -85,B 0,C 180,E1 -21858.002,E2 -21858.002} C_VEL
LIN {X 0,Y 342.605,Z 577.063,A -85,B 0,C 180,E1 -21859.941,E2 -21859.941} C_VEL
LIN {X 0,Y 347.435,Z 579.93,A -85,B 0,C 180,E1 -21862.38,E2 -21862.38} C_VEL
LIN {X 0,Y 350.433,Z 581.324,A -85,B 0,C 180,E1 -21864.245,E2 -21864.245} C_VEL
LIN {X 0,Y 352.333,Z 582.13,A -85,B 0,C 180,E1 -21865.819,E2 -21865.819} C_VEL
LIN {X 0,Y 353.137,Z 582.347,A -85,B 0,C 180,E1 -21866.577,E2 -21866.577} C_VEL
LIN {X 0,Y 353.906,Z 582.71,A -85,B 0,C 180,E1 -21867.723,E2 -21867.723} C_VEL
LIN {X 0,Y 354.31,Z 582.971,A -85,B 0,C 180,E1 -21868.863,E2 -21868.863} C_VEL
LIN {X 0,Y 354.549,Z 582.938,A -85,B 0,C 180,E1 -21870,E2 -21870} C_VEL
LIN {X 0,Y 354.351,Z 582.912,A -85,B 0,C 180,E1 -21871.136,E2 -21871.136} C_VEL
LIN {X 0,Y 353.905,Z 582.684,A -85,B 0,C 180,E1 -21872.276,E2 -21872.276} C_VEL
LIN {X 0,Y 352.34,Z 582.135,A -85,B 0,C 180,E1 -21874.198,E2 -21874.198} C_VEL
LIN {X 0,Y 350.373,Z 581.338,A -85,B 0,C 180,E1 -21875.756,E2 -21875.756} C_VEL
LIN {X 0,Y 347.448,Z 579.918,A -85,B 0,C 180,E1 -21877.636,E2 -21877.636} C_VEL
LIN {X 0,Y 342.6,Z 577.088,A -85,B 0,C 180,E1 -21880.054,E2 -21880.054} C_VEL
LIN {X 0,Y 338.075,Z 573.764,A -85,B 0,C 180,E1 -21881.998,E2 -21881.998} C_VEL
LIN {X 0,Y 334.16,Z 571.24,A -85,B 0,C 180,E1 -21883.376,E2 -21883.376} C_VEL
LIN {X 0,Y 327.825,Z 567.293,A -85,B 0,C 180,E1 -21885.267,E2 -21885.267} C_VEL
LIN {X 0,Y 322.769,Z 563.756,A -85,B 0,C 180,E1 -21886.656,E2 -21886.656} C_VEL
LIN {X 0,Y 316.919,Z 559.654,A -85,B 0,C 180,E1 -21888.087,E2 -21888.087} C_VEL
LIN {X 0,Y 309.69,Z 554.587,A -85,B 0,C 180,E1 -21889.651,E2 -21889.651} C_VEL
LIN {X 0,Y 304.339,Z 550.505,A -85,B 0,C 180,E1 -21890.734,E2 -21890.734} C_VEL
LIN {X 0,Y 296.012,Z 544.368,A -85,B 0,C 180,E1 -21892.191,E2 -21892.191} C_VEL
LIN {X 0,Y 281.46,Z 533.073,A -85,B 0,C 180,E1 -21894.581,E2 -21894.581} C_VEL
LIN {X 0,Y 269.81,Z 523.025,A -85,B 0,C 180,E1 -21896.547,E2 -21896.547} C_VEL
LIN {X 0,Y 259.457,Z 513.067,A -85,B 0,C 180,E1 -21898.319,E2 -21898.319} C_VEL
LIN {X 0,Y 247.772,Z 500.546,A -85,B 0,C 180,E1 -21900.307,E2 -21900.307} C_VEL
LIN {X 0,Y 237.104,Z 487.211,A -85,B 0,C 180,E1 -21902.305,E2 -21902.305} C_VEL
LIN {X 0,Y 228.87,Z 474.663,A -85,B 0,C 180,E1 -21904.094,E2 -21904.094} C_VEL
LIN {X 0,Y 222.008,Z 462.012,A -85,B 0,C 180,E1 -21905.804,E2 -21905.804} C_VEL
LIN {X 0,Y 214.796,Z 446.954,A -85,B 0,C 180,E1 -21907.838,E2 -21907.838} C_VEL
LIN {X 0,Y 207.369,Z 433.3,A -85,B 0,C 180,E1 -21910.066,E2 -21910.066} C_VEL
LIN {X 0,Y 199.964,Z 421.802,A -85,B 0,C 180,E1 -21912.434,E2 -21912.434} C_VEL
LIN {X 0,Y 197.671,Z 418.487,A -85,B 0,C 180,E1 -21913.211,E2 -21913.211} C_VEL
LIN {X 0,Y 195.25,Z 414.777,A -85,B 0,C 180,E1 -21914.073,E2 -21914.073} C_VEL
LIN {X 0,Y 193.322,Z 412.372,A -85,B 0,C 180,E1 -21914.757,E2 -21914.757} C_VEL
LIN {X 0,Y 192.643,Z 410.444,A -85,B 0,C 180,E1 -21915.248,E2 -21915.248} C_VEL
LIN {X 0,Y 192.54,Z 409.996,A -85,B 0,C 180,E1 -21916.092,E2 -21916.092} C_VEL
LIN {X 0,Y 192.55,Z 409.979,A -85,B 0,C 180,E1 -21920.038,E2 -21920.038} C_VEL
LIN {X 0,Y 192.596,Z 409.97,A -85,B 0,C 180,E1 -21924.279,E2 -21924.279} C_VEL
LIN {X 0,Y 192.603,Z 409.993,A -85,B 0,C 180,E1 -21929.281,E2 -21929.281} C_VEL
LIN {X 0,Y 192.66,Z 409.952,A -85,B 0,C 180,E1 -21931.693,E2 -21931.693} C_VEL
LIN {X 0,Y 192.701,Z 409.982,A -85,B 0,C 180,E1 -21936.349,E2 -21936.349} C_VEL
LIN {X 0,Y 192.727,Z 409.935,A -85,B 0,C 180,E1 -21941.459,E2 -21941.459} C_VEL
LIN {X 0,Y 192.768,Z 409.973,A -85,B 0,C 180,E1 -21945.215,E2 -21945.215} C_VEL
LIN {X 0,Y 192.977,Z 409.897,A -85,B 0,C 180,E1 -21949.509,E2 -21949.509} C_VEL
LIN {X 0,Y 193.064,Z 409.896,A -85,B 0,C 180,E1 -21951.629,E2 -21951.629} C_VEL
LIN {X 0,Y 193.261,Z 409.869,A -85,B 0,C 180,E1 -21957.917,E2 -21957.917} C_VEL
LIN {X 0,Y 193.437,Z 409.837,A -85,B 0,C 180,E1 -21960.001,E2 -21960.001} C_VEL
LIN {X 0,Y 192.976,Z 409.947,A -85,B 0,C 180,E1 -21964.178,E2 -21964.178} C_VEL
LIN {X 0,Y 193.059,Z 409.887,A -85,B 0,C 180,E1 -21968.374,E2 -21968.374} C_VEL
LIN {X 0,Y 192.85,Z 409.947,A -85,B 0,C 180,E1 -21972.631,E2 -21972.631} C_VEL
LIN {X 0,Y 192.755,Z 409.935,A -85,B 0,C 180,E1 -21976.96,E2 -21976.96} C_VEL
LIN {X 0,Y 192.635,Z 409.972,A -85,B 0,C 180,E1 -21981.399,E2 -21981.399} C_VEL
LIN {X 0,Y 192.663,Z 409.969,A -85,B 0,C 180,E1 -21984.226,E2 -21984.226} C_VEL
LIN {X 0,Y 192.649,Z 409.966,A -85,B 0,C 180,E1 -21988.894,E2 -21988.894} C_VEL
LIN {X 0,Y 192.599,Z 409.965,A -85,B 0,C 180,E1 -21993.187,E2 -21993.187} C_VEL
LIN {X 0,Y 192.6,Z 409.982,A -85,B 0,C 180,E1 -21998.342,E2 -21998.342} C_VEL
LIN {X 0,Y 192.677,Z 410.217,A -85,B 0,C 180,E1 -22001.914,E2 -22001.914} C_VEL
LIN {X 0,Y 193.588,Z 413.979,A -85,B 0,C 180,E1 -22004.884,E2 -22004.884} C_VEL
LIN {X 0,Y 195.677,Z 418.047,A -85,B 0,C 180,E1 -22005.825,E2 -22005.825} C_VEL
LIN {X 0,Y 197.532,Z 421.207,A -85,B 0,C 180,E1 -22006.497,E2 -22006.497} C_VEL
LIN {X 0,Y 202.52,Z 429.915,A -85,B 0,C 180,E1 -22008.219,E2 -22008.219} C_VEL
LIN {X 0,Y 208.043,Z 440.761,A -85,B 0,C 180,E1 -22010.034,E2 -22010.034} C_VEL
LIN {X 0,Y 214.831,Z 456.361,A -85,B 0,C 180,E1 -22012.173,E2 -22012.173} C_VEL
LIN {X 0,Y 216.007,Z 459.964,A -85,B 0,C 180,E1 -22012.561,E2 -22012.561} C_VEL
LIN {X 0,Y 218.408,Z 475.648,A -85,B 0,C 180,E1 -22013.666,E2 -22013.666} C_VEL
LIN {X 0,Y 216.269,Z 520.434,A -85,B 0,C 180,E1 -22015.105,E2 -22015.105} C_VEL
LIN {X 0,Y 215.262,Z 530.842,A -85,B 0,C 180,E1 -22015.634,E2 -22015.634} C_VEL
LIN {X 0,Y 213.869,Z 540.612,A -85,B 0,C 180,E1 -22016.323,E2 -22016.323} C_VEL
LIN {X 0,Y 212.232,Z 549.702,A -85,B 0,C 180,E1 -22017.164,E2 -22017.164} C_VEL
LIN {X 0,Y 210.247,Z 558.842,A -85,B 0,C 180,E1 -22018.233,E2 -22018.233} C_VEL
LIN {X 0,Y 208.043,Z 567.841,A -85,B 0,C 180,E1 -22019.555,E2 -22019.555} C_VEL
LIN {X 0,Y 205.593,Z 576.563,A -85,B 0,C 180,E1 -22021.129,E2 -22021.129} C_VEL
LIN {X 0,Y 203.322,Z 583.981,A -85,B 0,C 180,E1 -22022.743,E2 -22022.743} C_VEL
LIN {X 0,Y 200.4,Z 592.773,A -85,B 0,C 180,E1 -22025.114,E2 -22025.114} C_VEL
LIN {X 0,Y 198.135,Z 599.768,A -85,B 0,C 180,E1 -22027.456,E2 -22027.456} C_VEL
LIN {X 0,Y 196.241,Z 605.076,A -85,B 0,C 180,E1 -22029.564,E2 -22029.564} C_VEL
LIN {X 0,Y 195.356,Z 607.59,A -85,B 0,C 180,E1 -22030.728,E2 -22030.728} C_VEL
LIN {X 0,Y 193.683,Z 610.575,A -85,B 0,C 180,E1 -22032.152,E2 -22032.152} C_VEL
LIN {X 0,Y 189.357,Z 614.783,A -85,B 0,C 180,E1 -22034.506,E2 -22034.506} C_VEL
LIN {X 0,Y 185.285,Z 618.35,A -85,B 0,C 180,E1 -22037.063,E2 -22037.063} C_VEL
LIN {X 0,Y 184.051,Z 620.084,A -85,B 0,C 180,E1 -22038.765,E2 -22038.765} C_VEL
LIN {X 0,Y 183.214,Z 623.664,A -85,B 0,C 180,E1 -22043.393,E2 -22043.393} C_VEL
LIN {X 0,Y 183.056,Z 624.993,A -85,B 0,C 180,E1 -22046.587,E2 -22046.587} C_VEL
LIN {X 0,Y 183.15,Z 625.479,A -85,B 0,C 180,E1 -22050.001,E2 -22050.001} C_VEL
LIN {X 0,Y 183.035,Z 625.024,A -85,B 0,C 180,E1 -22053.301,E2 -22053.301} C_VEL
LIN {X 0,Y 183.181,Z 623.662,A -85,B 0,C 180,E1 -22056.61,E2 -22056.61} C_VEL
LIN {X 0,Y 183.99,Z 620.307,A -85,B 0,C 180,E1 -22061.011,E2 -22061.011} C_VEL
LIN {X 0,Y 185.117,Z 616.675,A -85,B 0,C 180,E1 -22064.287,E2 -22064.287} C_VEL
LIN {X 0,Y 186.848,Z 611.942,A -85,B 0,C 180,E1 -22067.513,E2 -22067.513} C_VEL
LIN {X 0,Y 189.13,Z 605.97,A -85,B 0,C 180,E1 -22070.672,E2 -22070.672} C_VEL
LIN {X 0,Y 190.885,Z 601.547,A -85,B 0,C 180,E1 -22072.588,E2 -22072.588} C_VEL
LIN {X 0,Y 192.906,Z 595.696,A -85,B 0,C 180,E1 -22074.77,E2 -22074.77} C_VEL
LIN {X 0,Y 195.789,Z 587.481,A -85,B 0,C 180,E1 -22077.237,E2 -22077.237} C_VEL
LIN {X 0,Y 198.384,Z 579.657,A -85,B 0,C 180,E1 -22079.151,E2 -22079.151} C_VEL
LIN {X 0,Y 200.851,Z 571.577,A -85,B 0,C 180,E1 -22080.78,E2 -22080.78} C_VEL
LIN {X 0,Y 203.519,Z 561.82,A -85,B 0,C 180,E1 -22082.361,E2 -22082.361} C_VEL
LIN {X 0,Y 205.45,Z 553.431,A -85,B 0,C 180,E1 -22083.477,E2 -22083.477} C_VEL
LIN {X 0,Y 207.585,Z 542.93,A -85,B 0,C 180,E1 -22084.548,E2 -22084.548} C_VEL
LIN {X 0,Y 209.187,Z 532.837,A -85,B 0,C 180,E1 -22085.325,E2 -22085.325} C_VEL
LIN {X 0,Y 210.413,Z 521.97,A -85,B 0,C 180,E1 -22085.912,E2 -22085.912} C_VEL
LIN {X 0,Y 211.617,Z 499.095,A -85,B 0,C 180,E1 -22086.712,E2 -22086.712} C_VEL
LIN {X 0,Y 212.689,Z 476.764,A -85,B 0,C 180,E1 -22087.421,E2 -22087.421} C_VEL
LIN {X 0,Y 210.368,Z 461.54,A -85,B 0,C 180,E1 -22088.549,E2 -22088.549} C_VEL
LIN {X 0,Y 204.202,Z 446.834,A -85,B 0,C 180,E1 -22090.594,E2 -22090.594} C_VEL
LIN {X 0,Y 198.549,Z 435.292,A -85,B 0,C 180,E1 -22092.548,E2 -22092.548} C_VEL
LIN {X 0,Y 191.87,Z 423.312,A -85,B 0,C 180,E1 -22095.009,E2 -22095.009} C_VEL
LIN {X 0,Y 189.001,Z 418.41,A -85,B 0,C 180,E1 -22096.142,E2 -22096.142} C_VEL
LIN {X 0,Y 186.788,Z 414.927,A -85,B 0,C 180,E1 -22097.066,E2 -22097.066} C_VEL
LIN {X 0,Y 186.217,Z 413.527,A -85,B 0,C 180,E1 -22097.512,E2 -22097.512} C_VEL
LIN {X 0,Y 185.555,Z 410.923,A -85,B 0,C 180,E1 -22099.916,E2 -22099.916} C_VEL
LIN {X 0,Y 185.563,Z 410.872,A -85,B 0,C 180,E1 -22102.699,E2 -22102.699} C_VEL
LIN {X 0,Y 185.548,Z 410.854,A -85,B 0,C 180,E1 -22107.974,E2 -22107.974} C_VEL
LIN {X 0,Y 185.585,Z 410.854,A -85,B 0,C 180,E1 -22110.575,E2 -22110.575} C_VEL
LIN {X 0,Y 185.589,Z 410.842,A -85,B 0,C 180,E1 -22115.382,E2 -22115.382} C_VEL
LIN {X 0,Y 185.609,Z 410.823,A -85,B 0,C 180,E1 -22120.074,E2 -22120.074} C_VEL
LIN {X 0,Y 185.726,Z 410.835,A -85,B 0,C 180,E1 -22124.639,E2 -22124.639} C_VEL
LIN {X 0,Y 185.926,Z 410.776,A -85,B 0,C 180,E1 -22129.358,E2 -22129.358} C_VEL
LIN {X 0,Y 185.962,Z 410.795,A -85,B 0,C 180,E1 -22133.489,E2 -22133.489} C_VEL
LIN {X 0,Y 186.209,Z 410.759,A -85,B 0,C 180,E1 -22137.836,E2 -22137.836} C_VEL
LIN {X 0,Y 186.405,Z 410.712,A -85,B 0,C 180,E1 -22139.999,E2 -22139.999} C_VEL
LIN {X 0,Y 185.927,Z 410.819,A -85,B 0,C 180,E1 -22144.334,E2 -22144.334} C_VEL
LIN {X 0,Y 186.014,Z 410.769,A -85,B 0,C 180,E1 -22148.691,E2 -22148.691} C_VEL
LIN {X 0,Y 185.765,Z 410.826,A -85,B 0,C 180,E1 -22153.119,E2 -22153.119} C_VEL
LIN {X 0,Y 185.69,Z 410.818,A -85,B 0,C 180,E1 -22157.624,E2 -22157.624} C_VEL
LIN {X 0,Y 185.596,Z 410.853,A -85,B 0,C 180,E1 -22162.25,E2 -22162.25} C_VEL
LIN {X 0,Y 185.559,Z 410.834,A -85,B 0,C 180,E1 -22167.031,E2 -22167.031} C_VEL
LIN {X 0,Y 185.576,Z 410.846,A -85,B 0,C 180,E1 -22169.492,E2 -22169.492} C_VEL
LIN {X 0,Y 185.508,Z 410.848,A -85,B 0,C 180,E1 -22174.629,E2 -22174.629} C_VEL
LIN {X 0,Y 185.542,Z 410.869,A -85,B 0,C 180,E1 -22177.303,E2 -22177.303} C_VEL
LIN {X 0,Y 185.457,Z 410.976,A -85,B 0,C 180,E1 -22182.231,E2 -22182.231} C_VEL
LIN {X 0,Y 185.691,Z 412.017,A -85,B 0,C 180,E1 -22182.784,E2 -22182.784} C_VEL
LIN {X 0,Y 187.308,Z 414.835,A -85,B 0,C 180,E1 -22183.511,E2 -22183.511} C_VEL
LIN {X 0,Y 188.751,Z 416.218,A -85,B 0,C 180,E1 -22184.048,E2 -22184.048} C_VEL
LIN {X 0,Y 190.988,Z 419.719,A -85,B 0,C 180,E1 -22184.926,E2 -22184.926} C_VEL
LIN {X 0,Y 192.215,Z 421.418,A -85,B 0,C 180,E1 -22185.382,E2 -22185.382} C_VEL
LIN {X 0,Y 197.671,Z 429.504,A -85,B 0,C 180,E1 -22187.326,E2 -22187.326} C_VEL
LIN {X 0,Y 205.182,Z 441.927,A -85,B 0,C 180,E1 -22189.805,E2 -22189.805} C_VEL
LIN {X 0,Y 212.941,Z 457.055,A -85,B 0,C 180,E1 -22192.195,E2 -22192.195} C_VEL
LIN {X 0,Y 221.146,Z 474.115,A -85,B 0,C 180,E1 -22194.509,E2 -22194.509} C_VEL
LIN {X 0,Y 229.553,Z 487.835,A -85,B 0,C 180,E1 -22196.509,E2 -22196.509} C_VEL
LIN {X 0,Y 238.216,Z 499.581,A -85,B 0,C 180,E1 -22198.296,E2 -22198.296} C_VEL
LIN {X 0,Y 249.19,Z 512.282,A -85,B 0,C 180,E1 -22200.342,E2 -22200.342} C_VEL
LIN {X 0,Y 260.857,Z 524.384,A -85,B 0,C 180,E1 -22202.546,E2 -22202.546} C_VEL
LIN {X 0,Y 272.198,Z 534.629,A -85,B 0,C 180,E1 -22204.644,E2 -22204.644} C_VEL
LIN {X 0,Y 286.101,Z 545.571,A -85,B 0,C 180,E1 -22207.097,E2 -22207.097} C_VEL
LIN {X 0,Y 297.24,Z 553.969,A -85,B 0,C 180,E1 -22209.058,E2 -22209.058} C_VEL
LIN {X 0,Y 302.729,Z 558.008,A -85,B 0,C 180,E1 -22210.087,E2 -22210.087} C_VEL
LIN {X 0,Y 310.739,Z 563.817,A -85,B 0,C 180,E1 -22211.787,E2 -22211.787} C_VEL
LIN {X 0,Y 316.878,Z 568.091,A -85,B 0,C 180,E1 -22213.242,E2 -22213.242} C_VEL
LIN {X 0,Y 322.769,Z 572.303,A -85,B 0,C 180,E1 -22214.853,E2 -22214.853} C_VEL
LIN {X 0,Y 327.95,Z 575.509,A -85,B 0,C 180,E1 -22216.365,E2 -22216.365} C_VEL
LIN {X 0,Y 332.256,Z 578.21,A -85,B 0,C 180,E1 -22217.788,E2 -22217.788} C_VEL
LIN {X 0,Y 336.068,Z 581.016,A -85,B 0,C 180,E1 -22219.379,E2 -22219.379} C_VEL
LIN {X 0,Y 338.434,Z 582.57,A -85,B 0,C 180,E1 -22220.437,E2 -22220.437} C_VEL
LIN {X 0,Y 340.984,Z 584.108,A -85,B 0,C 180,E1 -22221.704,E2 -22221.704} C_VEL
LIN {X 0,Y 343.24,Z 585.308,A -85,B 0,C 180,E1 -22222.943,E2 -22222.943} C_VEL
LIN {X 0,Y 345.856,Z 586.531,A -85,B 0,C 180,E1 -22224.682,E2 -22224.682} C_VEL
LIN {X 0,Y 347.983,Z 587.304,A -85,B 0,C 180,E1 -22226.526,E2 -22226.526} C_VEL
LIN {X 0,Y 348.8,Z 587.664,A -85,B 0,C 180,E1 -22227.69,E2 -22227.69} C_VEL
LIN {X 0,Y 349.238,Z 587.916,A -85,B 0,C 180,E1 -22228.847,E2 -22228.847} C_VEL
LIN {X 0,Y 349.478,Z 587.908,A -85,B 0,C 180,E1 -22230,E2 -22230} C_VEL
LIN {X 0,Y 349.273,Z 587.869,A -85,B 0,C 180,E1 -22231.153,E2 -22231.153} C_VEL
LIN {X 0,Y 348.793,Z 587.643,A -85,B 0,C 180,E1 -22232.309,E2 -22232.309} C_VEL
LIN {X 0,Y 347.959,Z 587.289,A -85,B 0,C 180,E1 -22233.473,E2 -22233.473} C_VEL
LIN {X 0,Y 345.857,Z 586.57,A -85,B 0,C 180,E1 -22235.321,E2 -22235.321} C_VEL
LIN {X 0,Y 343.207,Z 585.301,A -85,B 0,C 180,E1 -22237.057,E2 -22237.057} C_VEL
LIN {X 0,Y 340.929,Z 584.062,A -85,B 0,C 180,E1 -22238.322,E2 -22238.322} C_VEL
LIN {X 0,Y 338.413,Z 582.561,A -85,B 0,C 180,E1 -22239.563,E2 -22239.563} C_VEL
LIN {X 0,Y 334.463,Z 579.816,A -85,B 0,C 180,E1 -22241.329,E2 -22241.329} C_VEL
LIN {X 0,Y 331.243,Z 577.503,A -85,B 0,C 180,E1 -22242.586,E2 -22242.586} C_VEL
LIN {X 0,Y 325.252,Z 573.887,A -85,B 0,C 180,E1 -22244.44,E2 -22244.44} C_VEL
LIN {X 0,Y 318.54,Z 569.298,A -85,B 0,C 180,E1 -22246.317,E2 -22246.317} C_VEL
LIN {X 0,Y 313.299,Z 565.576,A -85,B 0,C 180,E1 -22247.635,E2 -22247.635} C_VEL
LIN {X 0,Y 305.407,Z 560.084,A -85,B 0,C 180,E1 -22249.357,E2 -22249.357} C_VEL
LIN {X 0,Y 298.881,Z 555.167,A -85,B 0,C 180,E1 -22250.653,E2 -22250.653} C_VEL
LIN {X 0,Y 286.093,Z 545.611,A -85,B 0,C 180,E1 -22252.9,E2 -22252.9} C_VEL
LIN {X 0,Y 272.207,Z 534.578,A -85,B 0,C 180,E1 -22255.36,E2 -22255.36} C_VEL
LIN {X 0,Y 258.973,Z 522.589,A -85,B 0,C 180,E1 -22257.809,E2 -22257.809} C_VEL
LIN {X 0,Y 247.811,Z 510.747,A -85,B 0,C 180,E1 -22259.918,E2 -22259.918} C_VEL
LIN {X 0,Y 236.888,Z 497.988,A -85,B 0,C 180,E1 -22261.96,E2 -22261.96} C_VEL
LIN {X 0,Y 226.713,Z 483.585,A -85,B 0,C 180,E1 -22264.13,E2 -22264.13} C_VEL
LIN {X 0,Y 219.073,Z 470.12,A -85,B 0,C 180,E1 -22266.04,E2 -22266.04} C_VEL
LIN {X 0,Y 209.546,Z 450.186,A -85,B 0,C 180,E1 -22268.83,E2 -22268.83} C_VEL
LIN {X 0,Y 202.607,Z 437.47,A -85,B 0,C 180,E1 -22271.023,E2 -22271.023} C_VEL
LIN {X 0,Y 195.427,Z 426.106,A -85,B 0,C 180,E1 -22273.457,E2 -22273.457} C_VEL
LIN {X 0,Y 190.993,Z 419.693,A -85,B 0,C 180,E1 -22275.074,E2 -22275.074} C_VEL
LIN {X 0,Y 188.775,Z 416.237,A -85,B 0,C 180,E1 -22275.943,E2 -22275.943} C_VEL
LIN {X 0,Y 186.377,Z 413.514,A -85,B 0,C 180,E1 -22276.866,E2 -22276.866} C_VEL
LIN {X 0,Y 185.615,Z 411.546,A -85,B 0,C 180,E1 -22277.347,E2 -22277.347} C_VEL
LIN {X 0,Y 185.493,Z 410.913,A -85,B 0,C 180,E1 -22277.928,E2 -22277.928} C_VEL
LIN {X 0,Y 185.539,Z 410.87,A -85,B 0,C 180,E1 -22282.696,E2 -22282.696} C_VEL
LIN {X 0,Y 185.54,Z 410.866,A -85,B 0,C 180,E1 -22287.976,E2 -22287.976} C_VEL
LIN {X 0,Y 185.577,Z 410.845,A -85,B 0,C 180,E1 -22290.576,E2 -22290.576} C_VEL
LIN {X 0,Y 185.583,Z 410.858,A -85,B 0,C 180,E1 -22295.383,E2 -22295.383} C_VEL
LIN {X 0,Y 185.67,Z 410.812,A -85,B 0,C 180,E1 -22301.134,E2 -22301.134} C_VEL
LIN {X 0,Y 185.72,Z 410.849,A -85,B 0,C 180,E1 -22304.641,E2 -22304.641} C_VEL
LIN {X 0,Y 185.92,Z 410.775,A -85,B 0,C 180,E1 -22309.36,E2 -22309.36} C_VEL
LIN {X 0,Y 185.962,Z 410.811,A -85,B 0,C 180,E1 -22313.491,E2 -22313.491} C_VEL
LIN {X 0,Y 186.205,Z 410.747,A -85,B 0,C 180,E1 -22317.838,E2 -22317.838} C_VEL
LIN {X 0,Y 186.401,Z 410.712,A -85,B 0,C 180,E1 -22320.001,E2 -22320.001} C_VEL
LIN {X 0,Y 185.924,Z 410.826,A -85,B 0,C 180,E1 -22324.337,E2 -22324.337} C_VEL
LIN {X 0,Y 186.006,Z 410.763,A -85,B 0,C 180,E1 -22328.694,E2 -22328.694} C_VEL
LIN {X 0,Y 185.762,Z 410.836,A -85,B 0,C 180,E1 -22333.122,E2 -22333.122} C_VEL
LIN {X 0,Y 185.688,Z 410.808,A -85,B 0,C 180,E1 -22337.626,E2 -22337.626} C_VEL
LIN {X 0,Y 185.595,Z 410.862,A -85,B 0,C 180,E1 -22342.253,E2 -22342.253} C_VEL
LIN {X 0,Y 185.561,Z 410.831,A -85,B 0,C 180,E1 -22347.034,E2 -22347.034} C_VEL
LIN {X 0,Y 185.578,Z 410.856,A -85,B 0,C 180,E1 -22349.495,E2 -22349.495} C_VEL
LIN {X 0,Y 185.52,Z 410.846,A -85,B 0,C 180,E1 -22354.629,E2 -22354.629} C_VEL
LIN {X 0,Y 185.568,Z 410.871,A -85,B 0,C 180,E1 -22357.315,E2 -22357.315} C_VEL
LIN {X 0,Y 185.564,Z 411.024,A -85,B 0,C 180,E1 -22360.323,E2 -22360.323} C_VEL
LIN {X 0,Y 186.323,Z 413.757,A -85,B 0,C 180,E1 -22362.61,E2 -22362.61} C_VEL
LIN {X 0,Y 188.764,Z 418.165,A -85,B 0,C 180,E1 -22363.77,E2 -22363.77} C_VEL
LIN {X 0,Y 190.212,Z 420.562,A -85,B 0,C 180,E1 -22364.347,E2 -22364.347} C_VEL
LIN {X 0,Y 193.768,Z 426.732,A -85,B 0,C 180,E1 -22365.719,E2 -22365.719} C_VEL
LIN {X 0,Y 199.963,Z 437.893,A -85,B 0,C 180,E1 -22367.943,E2 -22367.943} C_VEL
LIN {X 0,Y 206.556,Z 452.237,A -85,B 0,C 180,E1 -22370.199,E2 -22370.199} C_VEL
LIN {X 0,Y 210.461,Z 461.874,A -85,B 0,C 180,E1 -22371.485,E2 -22371.485} C_VEL
LIN {X 0,Y 212.688,Z 476.776,A -85,B 0,C 180,E1 -22372.579,E2 -22372.579} C_VEL
LIN {X 0,Y 210.438,Z 521.025,A -85,B 0,C 180,E1 -22374.036,E2 -22374.036} C_VEL
LIN {X 0,Y 209.317,Z 531.55,A -85,B 0,C 180,E1 -22374.591,E2 -22374.591} C_VEL
LIN {X 0,Y 208.011,Z 540.418,A -85,B 0,C 180,E1 -22375.24,E2 -22375.24} C_VEL
LIN {X 0,Y 206.288,Z 549.506,A -85,B 0,C 180,E1 -22376.092,E2 -22376.092} C_VEL
LIN {X 0,Y 204.232,Z 558.647,A -85,B 0,C 180,E1 -22377.182,E2 -22377.182} C_VEL
LIN {X 0,Y 201.949,Z 567.646,A -85,B 0,C 180,E1 -22378.534,E2 -22378.534} C_VEL
LIN {X 0,Y 199.401,Z 576.368,A -85,B 0,C 180,E1 -22380.144,E2 -22380.144} C_VEL
LIN {X 0,Y 197.027,Z 583.785,A -85,B 0,C 180,E1 -22381.796,E2 -22381.796} C_VEL
LIN {X 0,Y 193.95,Z 592.577,A -85,B 0,C 180,E1 -22384.226,E2 -22384.226} C_VEL
LIN {X 0,Y 191.666,Z 599.112,A -85,B 0,C 180,E1 -22386.451,E2 -22386.451} C_VEL
LIN {X 0,Y 189.597,Z 604.881,A -85,B 0,C 180,E1 -22388.814,E2 -22388.814} C_VEL
LIN {X 0,Y 187.593,Z 610.155,A -85,B 0,C 180,E1 -22391.432,E2 -22391.432} C_VEL
LIN {X 0,Y 185.583,Z 615.247,A -85,B 0,C 180,E1 -22394.629,E2 -22394.629} C_VEL
LIN {X 0,Y 184.318,Z 619.217,A -85,B 0,C 180,E1 -22397.895,E2 -22397.895} C_VEL
LIN {X 0,Y 184.051,Z 620.084,A -85,B 0,C 180,E1 -22398.765,E2 -22398.765} C_VEL
LIN {X 0,Y 182.968,Z 621.709,A -85,B 0,C 180,E1 -22400.508,E2 -22400.508} C_VEL
LIN {X 0,Y 179.683,Z 623.634,A -85,B 0,C 180,E1 -22403.4,E2 -22403.4} C_VEL
LIN {X 0,Y 177.11,Z 624.578,A -85,B 0,C 180,E1 -22405.811,E2 -22405.811} C_VEL
LIN {X 0,Y 176.046,Z 625.013,A -85,B 0,C 180,E1 -22407.708,E2 -22407.708} C_VEL
LIN {X 0,Y 175.968,Z 625.081,A -85,B 0,C 180,E1 -22408.353,E2 -22408.353} C_VEL
LIN {X 0,Y 176.058,Z 625.285,A -85,B 0,C 180,E1 -22410.001,E2 -22410.001} C_VEL
LIN {X 0,Y 175.951,Z 624.9,A -85,B 0,C 180,E1 -22413.038,E2 -22413.038} C_VEL
LIN {X 0,Y 176.118,Z 623.467,A -85,B 0,C 180,E1 -22416.876,E2 -22416.876} C_VEL
LIN {X 0,Y 176.996,Z 620.111,A -85,B 0,C 180,E1 -22421.452,E2 -22421.452} C_VEL
LIN {X 0,Y 178.191,Z 616.479,A -85,B 0,C 180,E1 -22424.855,E2 -22424.855} C_VEL
LIN {X 0,Y 180.068,Z 611.746,A -85,B 0,C 180,E1 -22428.195,E2 -22428.195} C_VEL
LIN {X 0,Y 182.494,Z 605.775,A -85,B 0,C 180,E1 -22431.461,E2 -22431.461} C_VEL
LIN {X 0,Y 184.63,Z 600.443,A -85,B 0,C 180,E1 -22433.81,E2 -22433.81} C_VEL
LIN {X 0,Y 187.017,Z 593.94,A -85,B 0,C 180,E1 -22436.204,E2 -22436.204} C_VEL
LIN {X 0,Y 189.482,Z 587.285,A -85,B 0,C 180,E1 -22438.223,E2 -22438.223} C_VEL
LIN {X 0,Y 192.188,Z 579.461,A -85,B 0,C 180,E1 -22440.187,E2 -22440.187} C_VEL
LIN {X 0,Y 194.788,Z 571.382,A -85,B 0,C 180,E1 -22441.849,E2 -22441.849} C_VEL
LIN {X 0,Y 197.558,Z 561.625,A -85,B 0,C 180,E1 -22443.463,E2 -22443.463} C_VEL
LIN {X 0,Y 199.559,Z 553.236,A -85,B 0,C 180,E1 -22444.603,E2 -22444.603} C_VEL
LIN {X 0,Y 201.787,Z 542.735,A -85,B 0,C 180,E1 -22445.689,E2 -22445.689} C_VEL
LIN {X 0,Y 203.497,Z 532.307,A -85,B 0,C 180,E1 -22446.498,E2 -22446.498} C_VEL
LIN {X 0,Y 204.674,Z 521.966,A -85,B 0,C 180,E1 -22447.073,E2 -22447.073} C_VEL
LIN {X 0,Y 205.903,Z 500.489,A -85,B 0,C 180,E1 -22447.839,E2 -22447.839} C_VEL
LIN {X 0,Y 206.998,Z 477.346,A -85,B 0,C 180,E1 -22448.602,E2 -22448.602} C_VEL
LIN {X 0,Y 204.976,Z 464.28,A -85,B 0,C 180,E1 -22449.63,E2 -22449.63} C_VEL
LIN {X 0,Y 199.298,Z 450.54,A -85,B 0,C 180,E1 -22451.63,E2 -22451.63} C_VEL
LIN {X 0,Y 194.284,Z 440.003,A -85,B 0,C 180,E1 -22453.47,E2 -22453.47} C_VEL
LIN {X 0,Y 187.861,Z 428.255,A -85,B 0,C 180,E1 -22455.972,E2 -22455.972} C_VEL
LIN {X 0,Y 184.772,Z 423.031,A -85,B 0,C 180,E1 -22457.256,E2 -22457.256} C_VEL
LIN {X 0,Y 181.805,Z 418.288,A -85,B 0,C 180,E1 -22458.546,E2 -22458.546} C_VEL
LIN {X 0,Y 179.33,Z 414.456,A -85,B 0,C 180,E1 -22459.71,E2 -22459.71} C_VEL
LIN {X 0,Y 178.771,Z 413.036,A -85,B 0,C 180,E1 -22460.294,E2 -22460.294} C_VEL
LIN {X 0,Y 178.473,Z 411.814,A -85,B 0,C 180,E1 -22461.544,E2 -22461.544} C_VEL
LIN {X 0,Y 178.494,Z 411.72,A -85,B 0,C 180,E1 -22466.547,E2 -22466.547} C_VEL
LIN {X 0,Y 178.526,Z 411.743,A -85,B 0,C 180,E1 -22470.005,E2 -22470.005} C_VEL
LIN {X 0,Y 178.527,Z 411.714,A -85,B 0,C 180,E1 -22474.882,E2 -22474.882} C_VEL
LIN {X 0,Y 178.625,Z 411.686,A -85,B 0,C 180,E1 -22480.783,E2 -22480.783} C_VEL
LIN {X 0,Y 178.689,Z 411.723,A -85,B 0,C 180,E1 -22486.349,E2 -22486.349} C_VEL
LIN {X 0,Y 178.939,Z 411.64,A -85,B 0,C 180,E1 -22490.96,E2 -22490.96} C_VEL
LIN {X 0,Y 179.155,Z 411.637,A -85,B 0,C 180,E1 -22497.751,E2 -22497.751} C_VEL
LIN {X 0,Y 179.368,Z 411.587,A -85,B 0,C 180,E1 -22499.999,E2 -22499.999} C_VEL
LIN {X 0,Y 178.876,Z 411.699,A -85,B 0,C 180,E1 -22504.506,E2 -22504.506} C_VEL
LIN {X 0,Y 178.963,Z 411.643,A -85,B 0,C 180,E1 -22509.036,E2 -22509.036} C_VEL
LIN {X 0,Y 178.687,Z 411.717,A -85,B 0,C 180,E1 -22513.649,E2 -22513.649} C_VEL
LIN {X 0,Y 178.649,Z 411.688,A -85,B 0,C 180,E1 -22518.342,E2 -22518.342} C_VEL
LIN {X 0,Y 178.511,Z 411.749,A -85,B 0,C 180,E1 -22523.183,E2 -22523.183} C_VEL
LIN {X 0,Y 178.484,Z 411.716,A -85,B 0,C 180,E1 -22528.196,E2 -22528.196} C_VEL
LIN {X 0,Y 178.497,Z 411.75,A -85,B 0,C 180,E1 -22530.786,E2 -22530.786} C_VEL
LIN {X 0,Y 178.488,Z 411.722,A -85,B 0,C 180,E1 -22534.221,E2 -22534.221} C_VEL
LIN {X 0,Y 178.474,Z 411.912,A -85,B 0,C 180,E1 -22539.782,E2 -22539.782} C_VEL
LIN {X 0,Y 178.727,Z 412.956,A -85,B 0,C 180,E1 -22540.359,E2 -22540.359} C_VEL
LIN {X 0,Y 180.214,Z 415.642,A -85,B 0,C 180,E1 -22541.111,E2 -22541.111} C_VEL
LIN {X 0,Y 181.874,Z 417.197,A -85,B 0,C 180,E1 -22541.802,E2 -22541.802} C_VEL
LIN {X 0,Y 183.927,Z 420.508,A -85,B 0,C 180,E1 -22542.705,E2 -22542.705} C_VEL
LIN {X 0,Y 185.42,Z 422.312,A -85,B 0,C 180,E1 -22543.306,E2 -22543.306} C_VEL
LIN {X 0,Y 193.107,Z 433.623,A -85,B 0,C 180,E1 -22546.265,E2 -22546.265} C_VEL
LIN {X 0,Y 200.723,Z 446.484,A -85,B 0,C 180,E1 -22548.926,E2 -22548.926} C_VEL
LIN {X 0,Y 207.681,Z 460.271,A -85,B 0,C 180,E1 -22551.193,E2 -22551.193} C_VEL
LIN {X 0,Y 216.416,Z 478.635,A -85,B 0,C 180,E1 -22553.787,E2 -22553.787} C_VEL
LIN {X 0,Y 224.909,Z 492.626,A -85,B 0,C 180,E1 -22555.898,E2 -22555.898} C_VEL
LIN {X 0,Y 233.308,Z 504.127,A -85,B 0,C 180,E1 -22557.706,E2 -22557.706} C_VEL
LIN {X 0,Y 243.646,Z 516.434,A -85,B 0,C 180,E1 -22559.818,E2 -22559.818} C_VEL
LIN {X 0,Y 254.505,Z 528.093,A -85,B 0,C 180,E1 -22562.085,E2 -22562.085} C_VEL
LIN {X 0,Y 266.632,Z 539.21,A -85,B 0,C 180,E1 -22564.523,E2 -22564.523} C_VEL
LIN {X 0,Y 280.088,Z 549.812,A -85,B 0,C 180,E1 -22567.073,E2 -22567.073} C_VEL
LIN {X 0,Y 292.76,Z 559.146,A -85,B 0,C 180,E1 -22569.426,E2 -22569.426} C_VEL
LIN {X 0,Y 300.111,Z 564.62,A -85,B 0,C 180,E1 -22570.861,E2 -22570.861} C_VEL
LIN {X 0,Y 307.456,Z 569.798,A -85,B 0,C 180,E1 -22572.428,E2 -22572.428} C_VEL
LIN {X 0,Y 314.197,Z 574.655,A -85,B 0,C 180,E1 -22574.116,E2 -22574.116} C_VEL
LIN {X 0,Y 321.11,Z 579.234,A -85,B 0,C 180,E1 -22576.069,E2 -22576.069} C_VEL
LIN {X 0,Y 325.839,Z 582.081,A -85,B 0,C 180,E1 -22577.544,E2 -22577.544} C_VEL
LIN {X 0,Y 331.105,Z 585.886,A -85,B 0,C 180,E1 -22579.673,E2 -22579.673} C_VEL
LIN {X 0,Y 335.114,Z 588.397,A -85,B 0,C 180,E1 -22581.558,E2 -22581.558} C_VEL
LIN {X 0,Y 337.453,Z 589.687,A -85,B 0,C 180,E1 -22582.821,E2 -22582.821} C_VEL
LIN {X 0,Y 339.467,Z 590.661,A -85,B 0,C 180,E1 -22584.058,E2 -22584.058} C_VEL
LIN {X 0,Y 341.117,Z 591.407,A -85,B 0,C 180,E1 -22585.273,E2 -22585.273} C_VEL
LIN {X 0,Y 342.474,Z 591.882,A -85,B 0,C 180,E1 -22586.47,E2 -22586.47} C_VEL
LIN {X 0,Y 343.355,Z 592.241,A -85,B 0,C 180,E1 -22587.653,E2 -22587.653} C_VEL
LIN {X 0,Y 343.817,Z 592.496,A -85,B 0,C 180,E1 -22588.828,E2 -22588.828} C_VEL
LIN {X 0,Y 344.062,Z 592.501,A -85,B 0,C 180,E1 -22590,E2 -22590} C_VEL
LIN {X 0,Y 343.846,Z 592.459,A -85,B 0,C 180,E1 -22591.171,E2 -22591.171} C_VEL
LIN {X 0,Y 343.351,Z 592.22,A -85,B 0,C 180,E1 -22592.346,E2 -22592.346} C_VEL
LIN {X 0,Y 342.451,Z 591.869,A -85,B 0,C 180,E1 -22593.529,E2 -22593.529} C_VEL
LIN {X 0,Y 341.079,Z 591.398,A -85,B 0,C 180,E1 -22594.727,E2 -22594.727} C_VEL
LIN {X 0,Y 339.236,Z 590.573,A -85,B 0,C 180,E1 -22596.063,E2 -22596.063} C_VEL
LIN {X 0,Y 337.426,Z 589.68,A -85,B 0,C 180,E1 -22597.179,E2 -22597.179} C_VEL
LIN {X 0,Y 334.292,Z 587.928,A -85,B 0,C 180,E1 -22598.851,E2 -22598.851} C_VEL
LIN {X 0,Y 331.106,Z 585.88,A -85,B 0,C 180,E1 -22600.328,E2 -22600.328} C_VEL
LIN {X 0,Y 327.109,Z 582.946,A -85,B 0,C 180,E1 -22601.985,E2 -22601.985} C_VEL
LIN {X 0,Y 322.058,Z 579.828,A -85,B 0,C 180,E1 -22603.65,E2 -22603.65} C_VEL
LIN {X 0,Y 315.629,Z 575.607,A -85,B 0,C 180,E1 -22605.497,E2 -22605.497} C_VEL
LIN {X 0,Y 309.003,Z 570.874,A -85,B 0,C 180,E1 -22607.208,E2 -22607.208} C_VEL
LIN {X 0,Y 301.911,Z 566.005,A -85,B 0,C 180,E1 -22608.768,E2 -22608.768} C_VEL
LIN {X 0,Y 295.418,Z 561.091,A -85,B 0,C 180,E1 -22610.082,E2 -22610.082} C_VEL
LIN {X 0,Y 281.715,Z 551.047,A -85,B 0,C 180,E1 -22612.627,E2 -22612.627} C_VEL
LIN {X 0,Y 269.375,Z 541.371,A -85,B 0,C 180,E1 -22614.959,E2 -22614.959} C_VEL
LIN {X 0,Y 259.904,Z 533.134,A -85,B 0,C 180,E1 -22616.833,E2 -22616.833} C_VEL
LIN {X 0,Y 249.728,Z 523.072,A -85,B 0,C 180,E1 -22618.919,E2 -22618.919} C_VEL
LIN {X 0,Y 238.919,Z 511.031,A -85,B 0,C 180,E1 -22621.152,E2 -22621.152} C_VEL
LIN {X 0,Y 228.255,Z 497.538,A -85,B 0,C 180,E1 -22623.349,E2 -22623.349} C_VEL
LIN {X 0,Y 219.531,Z 484.098,A -85,B 0,C 180,E1 -22625.4,E2 -22625.4} C_VEL
LIN {X 0,Y 212.826,Z 471.598,A -85,B 0,C 180,E1 -22627.221,E2 -22627.221} C_VEL
LIN {X 0,Y 205.077,Z 454.959,A -85,B 0,C 180,E1 -22629.635,E2 -22629.635} C_VEL
LIN {X 0,Y 198.691,Z 442.855,A -85,B 0,C 180,E1 -22631.763,E2 -22631.763} C_VEL
LIN {X 0,Y 191.525,Z 431.309,A -85,B 0,C 180,E1 -22634.312,E2 -22634.312} C_VEL
LIN {X 0,Y 186.913,Z 424.614,A -85,B 0,C 180,E1 -22636.082,E2 -22636.082} C_VEL
LIN {X 0,Y 184.473,Z 421.051,A -85,B 0,C 180,E1 -22637.08,E2 -22637.08} C_VEL
LIN {X 0,Y 182.248,Z 417.897,A -85,B 0,C 180,E1 -22638.026,E2 -22638.026} C_VEL
LIN {X 0,Y 181.343,Z 416.639,A -85,B 0,C 180,E1 -22638.42,E2 -22638.42} C_VEL
LIN {X 0,Y 179.399,Z 414.461,A -85,B 0,C 180,E1 -22639.261,E2 -22639.261} C_VEL
LIN {X 0,Y 178.566,Z 412.318,A -85,B 0,C 180,E1 -22639.875,E2 -22639.875} C_VEL
LIN {X 0,Y 178.445,Z 411.786,A -85,B 0,C 180,E1 -22640.576,E2 -22640.576} C_VEL
LIN {X 0,Y 178.492,Z 411.721,A -85,B 0,C 180,E1 -22645.775,E2 -22645.775} C_VEL
LIN {X 0,Y 178.518,Z 411.732,A -85,B 0,C 180,E1 -22650.007,E2 -22650.007} C_VEL
LIN {X 0,Y 178.53,Z 411.726,A -85,B 0,C 180,E1 -22654.876,E2 -22654.876} C_VEL
LIN {X 0,Y 178.619,Z 411.689,A -85,B 0,C 180,E1 -22660.785,E2 -22660.785} C_VEL
LIN {X 0,Y 178.661,Z 411.718,A -85,B 0,C 180,E1 -22664.018,E2 -22664.018} C_VEL
LIN {X 0,Y 178.857,Z 411.655,A -85,B 0,C 180,E1 -22669.211,E2 -22669.211} C_VEL
LIN {X 0,Y 178.925,Z 411.681,A -85,B 0,C 180,E1 -22673.234,E2 -22673.234} C_VEL
LIN {X 0,Y 179.151,Z 411.626,A -85,B 0,C 180,E1 -22677.753,E2 -22677.753} C_VEL
LIN {X 0,Y 179.365,Z 411.588,A -85,B 0,C 180,E1 -22680.001,E2 -22680.001} C_VEL
LIN {X 0,Y 178.872,Z 411.705,A -85,B 0,C 180,E1 -22684.508,E2 -22684.508} C_VEL
LIN {X 0,Y 178.935,Z 411.641,A -85,B 0,C 180,E1 -22689.04,E2 -22689.04} C_VEL
LIN {X 0,Y 178.685,Z 411.723,A -85,B 0,C 180,E1 -22693.651,E2 -22693.651} C_VEL
LIN {X 0,Y 178.621,Z 411.687,A -85,B 0,C 180,E1 -22699.218,E2 -22699.218} C_VEL
LIN {X 0,Y 178.523,Z 411.715,A -85,B 0,C 180,E1 -22705.119,E2 -22705.119} C_VEL
LIN {X 0,Y 178.5,Z 411.751,A -85,B 0,C 180,E1 -22710.788,E2 -22710.788} C_VEL
LIN {X 0,Y 178.484,Z 411.721,A -85,B 0,C 180,E1 -22714.221,E2 -22714.221} C_VEL
LIN {X 0,Y 178.498,Z 411.854,A -85,B 0,C 180,E1 -22718.599,E2 -22718.599} C_VEL
LIN {X 0,Y 178.974,Z 413.582,A -85,B 0,C 180,E1 -22720.019,E2 -22720.019} C_VEL
LIN {X 0,Y 181.287,Z 417.587,A -85,B 0,C 180,E1 -22721.229,E2 -22721.229} C_VEL
LIN {X 0,Y 182.967,Z 420.01,A -85,B 0,C 180,E1 -22721.96,E2 -22721.96} C_VEL
LIN {X 0,Y 186.319,Z 425.642,A -85,B 0,C 180,E1 -22723.396,E2 -22723.396} C_VEL
LIN {X 0,Y 191.778,Z 435.353,A -85,B 0,C 180,E1 -22725.583,E2 -22725.583} C_VEL
LIN {X 0,Y 196.911,Z 445.228,A -85,B 0,C 180,E1 -22727.498,E2 -22727.498} C_VEL
LIN {X 0,Y 204.029,Z 461.719,A -85,B 0,C 180,E1 -22730.036,E2 -22730.036} C_VEL
LIN {X 0,Y 205.35,Z 465.805,A -85,B 0,C 180,E1 -22730.523,E2 -22730.523} C_VEL
LIN {X 0,Y 207.03,Z 478.128,A -85,B 0,C 180,E1 -22731.439,E2 -22731.439} C_VEL
LIN {X 0,Y 204.751,Z 520.217,A -85,B 0,C 180,E1 -22732.835,E2 -22732.835} C_VEL
LIN {X 0,Y 203.701,Z 530.481,A -85,B 0,C 180,E1 -22733.381,E2 -22733.381} C_VEL
LIN {X 0,Y 202.222,Z 540.223,A -85,B 0,C 180,E1 -22734.094,E2 -22734.094} C_VEL
LIN {X 0,Y 200.442,Z 549.312,A -85,B 0,C 180,E1 -22734.961,E2 -22734.961} C_VEL
LIN {X 0,Y 198.31,Z 558.452,A -85,B 0,C 180,E1 -22736.072,E2 -22736.072} C_VEL
LIN {X 0,Y 195.919,Z 567.45,A -85,B 0,C 180,E1 -22737.448,E2 -22737.448} C_VEL
LIN {X 0,Y 193.259,Z 576.173,A -85,B 0,C 180,E1 -22739.093,E2 -22739.093} C_VEL
LIN {X 0,Y 190.798,Z 583.59,A -85,B 0,C 180,E1 -22740.788,E2 -22740.788} C_VEL
LIN {X 0,Y 187.565,Z 592.382,A -85,B 0,C 180,E1 -22743.281,E2 -22743.281} C_VEL
LIN {X 0,Y 185.363,Z 598.372,A -85,B 0,C 180,E1 -22745.352,E2 -22745.352} C_VEL
LIN {X 0,Y 182.99,Z 604.686,A -85,B 0,C 180,E1 -22748.01,E2 -22748.01} C_VEL
LIN {X 0,Y 180.855,Z 609.959,A -85,B 0,C 180,E1 -22750.713,E2 -22750.713} C_VEL
LIN {X 0,Y 178.715,Z 615.051,A -85,B 0,C 180,E1 -22754.022,E2 -22754.022} C_VEL
LIN {X 0,Y 177.349,Z 619.021,A -85,B 0,C 180,E1 -22757.412,E2 -22757.412} C_VEL
LIN {X 0,Y 176.468,Z 621.963,A -85,B 0,C 180,E1 -22760.834,E2 -22760.834} C_VEL
LIN {X 0,Y 176.142,Z 623.468,A -85,B 0,C 180,E1 -22763.126,E2 -22763.126} C_VEL
LIN {X 0,Y 175.972,Z 625.002,A -85,B 0,C 180,E1 -22767.712,E2 -22767.712} C_VEL
LIN {X 0,Y 175.968,Z 625.081,A -85,B 0,C 180,E1 -22768.353,E2 -22768.353} C_VEL
LIN {X 0,Y 175.293,Z 625.251,A -85,B 0,C 180,E1 -22770.264,E2 -22770.264} C_VEL
LIN {X 0,Y 173.686,Z 625.024,A -85,B 0,C 180,E1 -22772.144,E2 -22772.144} C_VEL
LIN {X 0,Y 170.051,Z 623.818,A -85,B 0,C 180,E1 -22775.944,E2 -22775.944} C_VEL
LIN {X 0,Y 169.21,Z 622.82,A -85,B 0,C 180,E1 -22777.917,E2 -22777.917} C_VEL
LIN {X 0,Y 169.229,Z 622.38,A -85,B 0,C 180,E1 -22778.579,E2 -22778.579} C_VEL
LIN {X 0,Y 170.402,Z 618.824,A -85,B 0,C 180,E1 -22783.112,E2 -22783.112} C_VEL
LIN {X 0,Y 171.871,Z 614.853,A -85,B 0,C 180,E1 -22786.633,E2 -22786.633} C_VEL
LIN {X 0,Y 174.534,Z 608.834,A -85,B 0,C 180,E1 -22790.631,E2 -22790.631} C_VEL
LIN {X 0,Y 177.391,Z 602.175,A -85,B 0,C 180,E1 -22793.93,E2 -22793.93} C_VEL
LIN {X 0,Y 180.05,Z 595.304,A -85,B 0,C 180,E1 -22796.673,E2 -22796.673} C_VEL
LIN {X 0,Y 183.254,Z 587.09,A -85,B 0,C 180,E1 -22799.274,E2 -22799.274} C_VEL
LIN {X 0,Y 186.077,Z 579.266,A -85,B 0,C 180,E1 -22801.288,E2 -22801.288} C_VEL
LIN {X 0,Y 188.802,Z 571.187,A -85,B 0,C 180,E1 -22802.984,E2 -22802.984} C_VEL
LIN {X 0,Y 191.666,Z 561.43,A -85,B 0,C 180,E1 -22804.636,E2 -22804.636} C_VEL
LIN {X 0,Y 193.749,Z 553.041,A -85,B 0,C 180,E1 -22805.797,E2 -22805.797} C_VEL
LIN {X 0,Y 196.072,Z 542.54,A -85,B 0,C 180,E1 -22806.898,E2 -22806.898} C_VEL
LIN {X 0,Y 197.855,Z 531.883,A -85,B 0,C 180,E1 -22807.738,E2 -22807.738} C_VEL
LIN {X 0,Y 199.074,Z 521.338,A -85,B 0,C 180,E1 -22808.327,E2 -22808.327} C_VEL
LIN {X 0,Y 200.544,Z 496.709,A -85,B 0,C 180,E1 -22809.2,E2 -22809.2} C_VEL
LIN {X 0,Y 201.446,Z 478.518,A -85,B 0,C 180,E1 -22809.812,E2 -22809.812} C_VEL
LIN {X 0,Y 199.68,Z 466.999,A -85,B 0,C 180,E1 -22810.765,E2 -22810.765} C_VEL
LIN {X 0,Y 194.399,Z 454.009,A -85,B 0,C 180,E1 -22812.747,E2 -22812.747} C_VEL
LIN {X 0,Y 189.285,Z 443.123,A -85,B 0,C 180,E1 -22814.75,E2 -22814.75} C_VEL
LIN {X 0,Y 181.528,Z 428.91,A -85,B 0,C 180,E1 -22818.027,E2 -22818.027} C_VEL
LIN {X 0,Y 177.905,Z 423.167,A -85,B 0,C 180,E1 -22819.68,E2 -22819.68} C_VEL
LIN {X 0,Y 174.743,Z 418.275,A -85,B 0,C 180,E1 -22821.221,E2 -22821.221} C_VEL
LIN {X 0,Y 172.063,Z 414.762,A -85,B 0,C 180,E1 -22822.584,E2 -22822.584} C_VEL
LIN {X 0,Y 171.502,Z 413.151,A -85,B 0,C 180,E1 -22823.177,E2 -22823.177} C_VEL
LIN {X 0,Y 171.42,Z 412.623,A -85,B 0,C 180,E1 -22824.25,E2 -22824.25} C_VEL
LIN {X 0,Y 171.461,Z 412.628,A -85,B 0,C 180,E1 -22829.403,E2 -22829.403} C_VEL
LIN {X 0,Y 171.465,Z 412.589,A -85,B 0,C 180,E1 -22834.387,E2 -22834.387} C_VEL
LIN {X 0,Y 171.581,Z 412.562,A -85,B 0,C 180,E1 -22840.871,E2 -22840.871} C_VEL
LIN {X 0,Y 171.605,Z 412.606,A -85,B 0,C 180,E1 -22845.774,E2 -22845.774} C_VEL
LIN {X 0,Y 171.875,Z 412.519,A -85,B 0,C 180,E1 -22850.585,E2 -22850.585} C_VEL
LIN {X 0,Y 171.825,Z 412.582,A -85,B 0,C 180,E1 -22855.306,E2 -22855.306} C_VEL
LIN {X 0,Y 172.332,Z 412.463,A -85,B 0,C 180,E1 -22859.999,E2 -22859.999} C_VEL
LIN {X 0,Y 171.825,Z 412.579,A -85,B 0,C 180,E1 -22864.691,E2 -22864.691} C_VEL
LIN {X 0,Y 171.892,Z 412.521,A -85,B 0,C 180,E1 -22869.411,E2 -22869.411} C_VEL
LIN {X 0,Y 171.61,Z 412.606,A -85,B 0,C 180,E1 -22874.223,E2 -22874.223} C_VEL
LIN {X 0,Y 171.544,Z 412.57,A -85,B 0,C 180,E1 -22879.56,E2 -22879.56} C_VEL
LIN {X 0,Y 171.461,Z 412.599,A -85,B 0,C 180,E1 -22885.61,E2 -22885.61} C_VEL
LIN {X 0,Y 171.454,Z 412.622,A -85,B 0,C 180,E1 -22890.593,E2 -22890.593} C_VEL
LIN {X 0,Y 171.409,Z 412.677,A -85,B 0,C 180,E1 -22896.705,E2 -22896.705} C_VEL
LIN {X 0,Y 171.574,Z 413.552,A -85,B 0,C 180,E1 -22897.445,E2 -22897.445} C_VEL
LIN {X 0,Y 173.127,Z 416.462,A -85,B 0,C 180,E1 -22898.38,E2 -22898.38} C_VEL
LIN {X 0,Y 175.177,Z 418.463,A -85,B 0,C 180,E1 -22899.352,E2 -22899.352} C_VEL
LIN {X 0,Y 177.272,Z 421.685,A -85,B 0,C 180,E1 -22900.375,E2 -22900.375} C_VEL
LIN {X 0,Y 178.669,Z 423.358,A -85,B 0,C 180,E1 -22901.003,E2 -22901.003} C_VEL
LIN {X 0,Y 182.601,Z 429.042,A -85,B 0,C 180,E1 -22902.737,E2 -22902.737} C_VEL
LIN {X 0,Y 188.965,Z 438.425,A -85,B 0,C 180,E1 -22905.295,E2 -22905.295} C_VEL
LIN {X 0,Y 196.217,Z 450.915,A -85,B 0,C 180,E1 -22907.976,E2 -22907.976} C_VEL
LIN {X 0,Y 203.122,Z 464.876,A -85,B 0,C 180,E1 -22910.352,E2 -22910.352} C_VEL
LIN {X 0,Y 211.601,Z 482.935,A -85,B 0,C 180,E1 -22912.999,E2 -22912.999} C_VEL
LIN {X 0,Y 219.906,Z 496.846,A -85,B 0,C 180,E1 -22915.169,E2 -22915.169} C_VEL
LIN {X 0,Y 228.316,Z 508.682,A -85,B 0,C 180,E1 -22917.114,E2 -22917.114} C_VEL
